DATA_BLOCK "GDB_ActiveRecipe"   // DB24
TITLE = Active recipes (Modules D+E, dual-pallet, PSC-bound)
{ S7_Optimized_Access := 'TRUE' }
// SCARA Phase 2 Module D + E active-recipe DB (V3.0, 2026-05-23). Two pallet slots (recipe1 = LEFT, recipe2 = RIGHT), each a UDT_Recipe. PSC binds member-for-member to recipe1.* and recipe2.* from separate HMI parameter sets. Pallet selection is operator-driven via the maintained bo_ExecutePallet1 / bo_ExecutePallet2 flags (WanErXin pattern -- no auto-advance); FB_PatternAutoGen mediates the mutex, picks the active recipe, writes its config to GDB_PalletizingCmd, validates both recipes independently, and latches per-pallet bo_PalletNFull alarms on cycle completion attributed to the IN-FLIGHT pallet (snapshotted at cycle start, so mid-cycle operator swaps cannot mis-attribute). Operator swaps pallets by clearing one flag and setting the other -- the just-emptied side's full bit auto-clears so it can be re-used. V3.0 also adds explicit per-pallet bo_AckPalletNFull reset bits and the bo_BothPalletsFull aggregate for HMI / future module integration.
// stored: MemoryReserve 100
   VAR
      recipe1 : "UDT_Recipe";   // Active recipe for PALLET 1 (LEFT). PSC binds and writes here from the HMI's pallet-1 parameter set. FB_PatternAutoGen consumes this each scan iff recipe1.bo_Valid is TRUE AND i16_ActivePalletIdx = 1. StartValues = the verified 16-box 4x(2x2) Module D default.
      recipe2 : "UDT_Recipe";   // Active recipe for PALLET 2 (RIGHT). PSC binds and writes here from the HMI's pallet-2 parameter set. FB_PatternAutoGen consumes this each scan iff recipe2.bo_Valid is TRUE AND i16_ActivePalletIdx = 2. StartValues match recipe1 (pallets share a default product); operator overrides via PSC if pallet 2 should carry a different box product.
      bo_PatternValid1 : Bool;   // FB_PatternAutoGen status for PALLET 1: recipe1 passed validation and its computed grid is mathematically valid. HMI lamp. (Independent of whether pallet 1 is currently active.)
      bo_PatternValid2 : Bool;   // FB_PatternAutoGen status for PALLET 2: recipe2 passed validation.
      bo_PatternError1 : Bool;   // FB_PatternAutoGen status for PALLET 1: recipe1 failed validation. HMI alarm.
      bo_PatternError2 : Bool;   // FB_PatternAutoGen status for PALLET 2: recipe2 failed validation.
      i16_ComputedGridColsX1 : Int;   // FB_PatternAutoGen echo for PALLET 1: auto-fitted columns along X.
      i16_ComputedGridColsX2 : Int;   // FB_PatternAutoGen echo for PALLET 2: auto-fitted columns along X.
      i16_ComputedGridRowsY1 : Int;   // FB_PatternAutoGen echo for PALLET 1: auto-fitted rows along Y.
      i16_ComputedGridRowsY2 : Int;   // FB_PatternAutoGen echo for PALLET 2: auto-fitted rows along Y.
      i16_ComputedBoxCount1 : Int;   // FB_PatternAutoGen echo for PALLET 1: total boxes = Cols x Rows x LayerCount. Must stay within the GDB_PalletizingPath.aCmd[] ceiling (22) or recipe1 is rejected.
      i16_ComputedBoxCount2 : Int;   // FB_PatternAutoGen echo for PALLET 2: total boxes. Same ceiling.
      bo_ExecutePallet1 : Bool := TRUE;   // Operator flag (HMI MAINTAINED button) -- "execute pallet 1" (WanErXin pattern). Setting TRUE while bo_ExecutePallet2=FALSE selects pallet 1 as active; FB_PatternAutoGen then writes recipe1 into GDB_PalletizingCmd. Cleared TRUE by operator releasing the button OR auto-cleared by FB when bo_Pallet1Full (operator must press the other side's button to swap, which auto-clears the just-emptied pallet's full bit so it can be re-used).
      bo_ExecutePallet2 : Bool := FALSE;   // Operator flag -- "execute pallet 2". Mirror of bo_ExecutePallet1 for the right-side pallet. Both flags simultaneously TRUE = mutex stalemate (FB keeps the current active pallet); both FALSE = i16_ActivePalletIdx := 0, no pallet active, GDB_PalletizingCmd left at safe defaults.
      i16_ActivePalletIdx : Int;   // FB_PatternAutoGen status: which pallet is currently active. 1 = pallet 1 (LEFT), 2 = pallet 2 (RIGHT), 0 = neither (no operator flag set OR active recipe invalid). HMI display.
      bo_Pallet1Full : Bool;   // Latched "pallet 1 full" alarm. Set TRUE by FB_PatternAutoGen when GDB_PalletizingCmd.bo_PalletDone is TRUE while i16_ActivePalletIdx = 1 (the cycle just placed the last box of pallet 1). Cleared automatically when the operator switches to pallet 2 (bo_ExecutePallet1 := FALSE AND bo_ExecutePallet2 := TRUE) -- which is interpreted as "I have emptied pallet 1, ready to re-use it later". HMI lamp/alarm.
      bo_Pallet2Full : Bool;   // Latched "pallet 2 full" alarm. Same logic as bo_Pallet1Full, mirrored.
      bo_AckPallet1Full : Bool;   // V3.0 (2026-05-23): Operator acknowledge / explicit reset for bo_Pallet1Full. HMI MAINTAINED button. While TRUE, FB_PatternAutoGen forces bo_Pallet1Full := FALSE every scan -- explicit reset path used when operator has physically emptied pallet 1 and wants to re-use it WITHOUT first having to swap to pallet 2. (The WanErXin swap-clear path remains as a convenience: pressing pallet 2's button while pallet 1's full bit is latched still clears it.) Operator releases the Ack button before re-starting the cycle so the next bo_PalletDone can re-latch bo_Pallet1Full normally.
      bo_AckPallet2Full : Bool;   // V3.0: Operator acknowledge / explicit reset for bo_Pallet2Full. Mirror of bo_AckPallet1Full.
      bo_BothPalletsFull : Bool;   // V3.0: FB-computed aggregate = bo_Pallet1Full AND bo_Pallet2Full. Single status bit for HMI / future Module F-G integration to gate "both pallets need unloading, robot should idle". Read-only from HMI side -- FB_PatternAutoGen is sole writer.
   END_VAR
BEGIN
   recipe1.sName := 'Pallet 1 Default 4x2x2';
   recipe1.bo_Valid := TRUE;
   recipe1.product.lr_Length := 400.0;
   recipe1.product.lr_Width := 600.0;
   recipe1.product.lr_Height := 200.0;
   recipe1.product.lr_Gap := 0.0;
   recipe1.pallet.lr_BaseLength := 800.0;
   recipe1.pallet.lr_BaseWidth := 1200.0;
   recipe1.pallet.i16_LayerCount := 4;
   recipe1.dynamics.lr_Velocity := 2000.0;
   recipe1.dynamics.lr_Acceleration := 10000.0;
   recipe1.dynamics.lr_Deceleration := 10000.0;
   recipe1.dynamics.lr_Jerk := 100000.0;
   recipe2.sName := 'Pallet 2 Default 4x2x2';
   recipe2.bo_Valid := TRUE;
   recipe2.product.lr_Length := 400.0;
   recipe2.product.lr_Width := 600.0;
   recipe2.product.lr_Height := 200.0;
   recipe2.product.lr_Gap := 0.0;
   recipe2.pallet.lr_BaseLength := 800.0;
   recipe2.pallet.lr_BaseWidth := 1200.0;
   recipe2.pallet.i16_LayerCount := 4;
   recipe2.dynamics.lr_Velocity := 2000.0;
   recipe2.dynamics.lr_Acceleration := 10000.0;
   recipe2.dynamics.lr_Deceleration := 10000.0;
   recipe2.dynamics.lr_Jerk := 100000.0;
END_DATA_BLOCK

DATA_BLOCK "GDB_MovePath"   // DB21
{ S7_Optimized_Access := 'TRUE' }
// stored: MemoryReserve 100
BEGIN
END_DATA_BLOCK

DATA_BLOCK "GDB_TeachCmd"   // DB27
TITLE = Teach mode commands + status (Module F)
{ S7_Optimized_Access := 'TRUE' }
// SCARA Phase 2 Module F teach-mode command + status DB (2026-05-23). HMI writes the mode toggle, per-slot operations (Capture/Verify/Clear/ClearAll), and replay controls (Start/Stop/Vel). FB_TeachCtrl reads them, executes via the shared GDB_AxisCtrl interface, and publishes back i16_TeachStep / i16_ReplayIdx / bo_ReplayDone for HMI display. Mode mutex: bo_Mode must be TRUE while GDB_MachineCmd.bo_Mode (transitional), GDB_PalletizingCmd.bo_Mode, and GDB_ManualCmd.bo_Mode are all FALSE.
// stored: MemoryReserve 100
   VAR
      bo_Mode : Bool := FALSE;   // HMI: Teach mode selector (the 4th mutex mode). TRUE = teach commands + jog active and the replay FSM can run. FALSE = ignored. Mutex with GDB_MachineCmd.bo_Mode (ABCDE, transitional -- to be deleted), GDB_PalletizingCmd.bo_Mode (palletizing), GDB_ManualCmd.bo_Mode (manual). FB_TeachCtrl REGION Mode_Gate enforces single-mode-active via statTeachOK.
      bo_ESTOP_LOCK : Bool := TRUE;   // Safety: E-Stop chain healthy (TRUE = OK, FALSE = E-Stop active). Mirrors GDB_PalletizingCmd / GDB_ManualCmd convention. Default TRUE (PLCSIM phantom; real fieldbus E-Stop integration is a separate task).
      i16_SlotIdx : Int := 1;   // HMI: which teach slot (1..16) the operator is currently operating on. Used by all four edge-pulsed operations (Capture, Verify, Clear) and as the HMI's "table row selector". Validated by FB_TeachCtrl as 1 <= idx <= 16; out-of-range pulses are ignored. Default 1.
      bo_Capture : Bool;   // HMI PULSE: capture current TCP into aPoints[i16_SlotIdx]. Edge-detected by FB_TeachCtrl. On rising edge (and only while statTeachOK = TRUE AND idx in range): reads GDB_AxisCtrl.LKinCtrl.output.actualposition (populated by FB_AxisCtrl MirrorTCP from ScaraArm3D.Position[..]), writes to aPoints[idx].position[0..3] (4..5 zeroed), sets abCaptured[idx] := TRUE, sets i16_TeachStep := 10 briefly for HMI feedback. Operator's main teach action.
      bo_Verify : Bool;   // HMI PULSE: move robot to aPoints[i16_SlotIdx]. Edge-detected. On rising edge: copies aPoints[idx].position to GDB_AxisCtrl.LKinCtrl.input.movelinear.targetposition, sets r64_velocity to lr_ReplayVel, pulses bo_execute. Used to validate that a captured slot points where the operator intended.
      bo_Clear : Bool;   // HMI PULSE: clear aPoints[i16_SlotIdx] (zero the position fields) and set abCaptured[idx] := FALSE. Edge-detected. Operator re-arms the slot for capture.
      bo_ClearAll : Bool;   // HMI PULSE: clear ALL 16 slots in one pass. Edge-detected. FB loops 1..16 clearing both aPoints[i] and abCaptured[i]. Operator's "wipe and start over" gesture.
      bo_StartReplay : Bool;   // HMI PULSE: start once-through replay of all captured slots in index order. Edge-detected. FB_TeachCtrl Replay_FSM transitions from idle (0) to load_next_slot (100), iterates aPoints[1..16] skipping uncaptured slots, drives each via the shared movelinear interface. Replay ends with bo_ReplayDone := TRUE and FSM back to idle.
      bo_StopReplay : Bool;   // HMI PULSE: abort replay immediately. Edge-detected. FB_TeachCtrl Replay_FSM transitions to idle (0) from any active state, clears bo_execute, the current move aborts via the MC layer's bo_commandaborted.
      lr_ReplayVel : LReal := 200.0;   // HMI: replay-move velocity (mm/s). Applied uniformly to every replay move and to bo_Verify moves. Default 200.0 mm/s (matches FB_ManualCtrl's safe-jog Cartesian dynamic). Auto-cycle palletizing uses 300+ mm/s.
      i16_TeachStep : Int;   // FB status: current step in FB_TeachCtrl Operator_Actions / Replay_FSM. Values: 0=idle, 10=capture-pulse-handled, 20=verify-in-flight, 30=clear-applied, 100=replay-running (i16_ReplayIdx advancing), 200=replay-done (latched until next StartReplay), 800=fault. HMI status display.
      i16_ReplayIdx : Int;   // FB status: which slot is currently being executed during replay (1..16). 0 when idle. HMI highlights the active row in the teach-table view.
      bo_ReplayDone : Bool;   // FB status: latched TRUE when replay reaches the end of captured slots (once-through). Cleared on next bo_StartReplay rising edge or on mode exit. HMI displays as a "Replay complete" lamp.
   END_VAR
BEGIN
END_DATA_BLOCK

DATA_BLOCK "GDB_TeachPoints"   // DB26
TITLE = Teach-point storage (Module F, 16 slots)
{ S7_Optimized_Access := 'TRUE' }
// SCARA Phase 2 Module F teach-point storage (V1.1, 2026-05-23). 16 slots, each carrying BOTH Cartesian TCP (aPoints[i] = LKinCtrl_typePoint, Siemens-canonical) AND joint angles (aJointAngles[i] = Array[1..4] of LReal for J1-J4). V1.1 added joint capture per Phase 2 spec §7.1 ("捕获脉冲 → 当前 TCP/关节 写点表"). Operator captures both in one bo_Capture pulse via FB_TeachCtrl. Replay (bo_StartReplay) currently walks aPoints via Cartesian linear moves; joint-space PTP replay using aJointAngles is reserved for a future extension.
// stored: MemoryReserve 100
   VAR
      aPoints : Array[1..16] of "LKinCtrl_typePoint";   // Module F teach-point slots (1..16) -- CARTESIAN. Each slot reuses the Siemens-canonical LKinCtrl_typePoint UDT: name (WString), position[0..5] LReal (Cartesian X/Y/Z/A/B/C in WCS; SCARA populates [0..3] only), coordSystem USInt (default 0=WCS), linkConstellation DWord, turnJoint[0..5] DInt. FB_TeachCtrl writes here on operator's bo_Capture edge from GDB_AxisCtrl.LKinCtrl.output.actualposition. Replay (bo_StartReplay) walks these via Cartesian linear moves.
      aJointAngles : Array[1..16, 1..4] of LReal;   // V1.1 (2026-05-23, joint extension per Phase 2 §7.1 spec "TCP/关节"): Per-slot joint angles J1/J2/J3/J4 captured at the same scan as aPoints[i]. 2D array (S7-1500T does not allow nested Array-of-Array in interface declarations -- same convention LKinCtrl_FrameTransTool's rotation matrices use). Access: aJointAngles[slot, joint] e.g. aJointAngles[3, 1] = slot 3's J1. FB_TeachCtrl writes from "ScaraArm3D".AxesData.A[1..4].Position on the same bo_Capture rising edge. Stored for archival + future joint-space PTP replay (currently replay is Cartesian-linear only). J1/J2/J4 in degrees, J3 in mm (prismatic Z per the SCARA TO config).
      abCaptured : Array[1..16] of Bool;   // Per-slot "this slot has been captured" flag. FB_TeachCtrl sets TRUE on bo_Capture rising edge for slot i16_SlotIdx (one set covers BOTH aPoints[idx] and aJointAngles[idx], V1.1); clears on bo_Clear or bo_ClearAll. Replay (bo_StartReplay) skips slots where this is FALSE. Default FALSE (no slots captured at boot).
      i16_PointCount : Int;   // FB-computed status: COUNT of TRUE bits in abCaptured[1..16]. HMI displays as "Captured slots: N / 16". Also used by FB_TeachCtrl Replay_FSM as the bound for the slot iteration (replay only runs slots where abCaptured = TRUE).
   END_VAR
BEGIN
END_DATA_BLOCK

ORGANIZATION_BLOCK "Main"   // OB1, LAD, ProgramCycle
TITLE = "Main Program Sweep (Cycle)"
{ S7_Optimized_Access := 'TRUE' }
// stored: SetENOAutomatically false
   VAR_INPUT
      Initial_Call : Bool;   // Initial call of this OB
      Remanence : Bool;   // =True, if remanent data are available
   END_VAR
BEGIN
END_ORGANIZATION_BLOCK

ORGANIZATION_BLOCK "CyclicInterrupt_10ms"   // OB30, LAD, CyclicInterrupt
{ S7_Optimized_Access := 'TRUE' }
// stored: SetENOAutomatically false
   VAR_INPUT
      Initial_Call : Bool;   // Initial call of this OB
      Event_Count : Int;   // Events discarded
   END_VAR
BEGIN
END_ORGANIZATION_BLOCK

ORGANIZATION_BLOCK "Startup"
TITLE = "Complete Restart"
{ S7_Optimized_Access := 'TRUE' }
VERSION : 1.0
// =====================================================================
// SCARA ABCDE â€” Startup (OB100)
//
// 2026-05-17 â€” Minimal startup for ABCDE 5-point demo.
// Initializes GDB_Control arrays so retain-memory drift can never zero
// them (defense pattern proven in v9, see Memory MEMORY.md â†’ cfg-retain
// fix). Clears command bits so warm-start can't replay an in-flight cmd.
//
// All HMI cmd bits live in GDB_MachineCmd (initialized via Member
// StartValue attributes in the XML â€” bo_Mode and bo_ESTOP_LOCK both
// default TRUE so an operator can immediately start). i16_AutoStep
// defaults to 0 (idle) which is the safe state.
// =====================================================================
   VAR_TEMP 
      i : Int;
   END_VAR


BEGIN
	
	 REGION Set_GroupPower_StartStopMode_defaults
	     // LKinCtrl_MC_GroupPower reads GDB_Control.StartMode[i] / StopMode[i].
	     // If any element is 0 on cold start / warm-start retain drift, MC_Power
	     // silently refuses to assert axesEnabled  - busy stuck FALSE forever.
	     // Set all 6 elements of both arrays to 1 (position-controlled enable /
	     // standard immediate-stop) on every PLC startup.
	     FOR #i := 1 TO 6 DO
	         "GDB_AxisCtrl".LKinCtrl.input.configuration.power.startMode[#i] := 1;   // 1 = enable position-controlled
	         "GDB_AxisCtrl".LKinCtrl.input.configuration.power.stopMode[#i]  := 1;   // 1 = immediate stop
	     END_FOR;
	 END_REGION
	
	 REGION Set_GroupHome_defaults
	     // LKinCtrl_MC_GroupHome reads GDB_Control.HomePos[i] / HomeMode[i].
	     // HomeMode=7 ("set actual position") is used in the SCARA demo so
	     // no physical homing motion is needed  - the operator clicks Home
	     // and the current TO joint position becomes the home reference.
	     //
	     // HomePos values per kinematic-axis index (A1=J1 base, A2=J3 z,
	     // A3=J2 elbow, A4=J4 wrist) match the SCARA3D zero pose. Indexes
	     // 5/6 (B/C orientation) unused in this 4-DOF kinematic.
	     "GDB_AxisCtrl".LKinCtrl.input.configuration.home.r64_homeposition[1] := 0.0;   // A1 = J1 base shoulder
	     "GDB_AxisCtrl".LKinCtrl.input.configuration.home.r64_homeposition[2] := 0.0;   // A2 = J3 prismatic z
	     "GDB_AxisCtrl".LKinCtrl.input.configuration.home.r64_homeposition[3] := 0.0;   // A3 = J2 elbow
	     "GDB_AxisCtrl".LKinCtrl.input.configuration.home.r64_homeposition[4] := 0.0;   // A4 = J4 wrist
	     "GDB_AxisCtrl".LKinCtrl.input.configuration.home.r64_homeposition[5] := 0.0;   // unused
	     "GDB_AxisCtrl".LKinCtrl.input.configuration.home.r64_homeposition[6] := 0.0;   // unused
	     FOR #i := 1 TO 6 DO
	         "GDB_AxisCtrl".LKinCtrl.input.configuration.home.i16_mode[#i] := 7;   // 7 = set actual position (no motion)
	     END_FOR;
	 END_REGION
	
	 REGION Set_GroupReset_RestartMode_defaults
	     // LKinCtrl_MC_GroupReset reads GDB_Control.RestartMode[1..7] of Bool.
	     // All FALSE = standard reset (clear axis error, do not re-initialize TO).
	     FOR #i := 1 TO 7 DO
	         "GDB_AxisCtrl".LKinCtrl.input.configuration.reset.restart[#i] := FALSE;
	     END_FOR;
	 END_REGION
	
	 REGION Clear_group_motion_command_bits
	     // Defensive: clear group enable/home/reset bits so warm-start can't
	     // replay an in-flight command. Operator must re-click Enable on HMI.
	     "GDB_AxisCtrl".LKinCtrl.input.bo_enable := FALSE;
	     "GDB_AxisCtrl".LKinCtrl.input.bo_reset  := FALSE;
	     "GDB_AxisCtrl".LKinCtrl.input.bo_home   := FALSE;
	 END_REGION
	
	 REGION Clear_AutoCtrl_command_bits
	     // Wang Shuo pattern: i16_AutoStep is the master state. 0 = idle.
	     // On warm-start, retain may have left step=80 (mid-cycle). Force
	     // back to 0 so operator must explicitly re-Start.
	     "GDB_MachineCmd".i16_AutoStep := 0;
	     "GDB_MachineCmd".bo_PathInitialed := FALSE;  // operator must re-init
	     "GDB_MachineCmd".bo_Alarm := FALSE;
	 END_REGION
	
	 REGION Clear_PalletizingCtrl_command_bits
	     // C69 Phase 2.2 (2026-05-18): defensively clear all palletizing-mode
	     // command bits + i16_PalletStep so warm-start can't replay a partial
	     // cycle. bo_Mode + bo_ESTOP_LOCK keep their XML StartValues (FALSE + TRUE).
	     // bo_PalletInitialed cleared - operator must re-pulse bo_InitPallet on
	     // session start to repopulate pts[] (path table is in iDB statics, not
	     // retain, so it would be all-zeros after memory reset anyway).
	     "GDB_PalletizingCmd".bo_InitPallet := FALSE;
	     "GDB_PalletizingCmd".bo_Start := FALSE;
	     "GDB_PalletizingCmd".bo_Stop := FALSE;
	     "GDB_PalletizingCmd".bo_PalletInitialed := FALSE;
	     "GDB_PalletizingCmd".bo_Alarm := FALSE;
	     "GDB_PalletizingCmd".i16_PalletStep := 0;
	 END_REGION
	
	 REGION Clear_ManualCtrl_command_bits
	     // Phase G (C67, 2026-05-18): defensively clear all manual-mode
	     // command bits so warm-start can't replay a held jog button or
	     // a latched Enable/Home/Reset. Operator must re-press on HMI.
	     // bo_Mode + bo_ESTOP_LOCK keep their XML StartValues (FALSE + TRUE).
	     "GDB_ManualCmd".bo_J1_Enable := FALSE;
	     "GDB_ManualCmd".bo_J2_Enable := FALSE;
	     "GDB_ManualCmd".bo_J3_Enable := FALSE;
	     "GDB_ManualCmd".bo_J4_Enable := FALSE;
	     "GDB_ManualCmd".bo_J1_Home := FALSE;
	     "GDB_ManualCmd".bo_J2_Home := FALSE;
	     "GDB_ManualCmd".bo_J3_Home := FALSE;
	     "GDB_ManualCmd".bo_J4_Home := FALSE;
	     "GDB_ManualCmd".bo_J1_Reset := FALSE;
	     "GDB_ManualCmd".bo_J2_Reset := FALSE;
	     "GDB_ManualCmd".bo_J3_Reset := FALSE;
	     "GDB_ManualCmd".bo_J4_Reset := FALSE;
	     "GDB_ManualCmd".bo_J1_JogForward := FALSE;
	     "GDB_ManualCmd".bo_J1_JogBackward := FALSE;
	     "GDB_ManualCmd".bo_J2_JogForward := FALSE;
	     "GDB_ManualCmd".bo_J2_JogBackward := FALSE;
	     "GDB_ManualCmd".bo_J3_JogForward := FALSE;
	     "GDB_ManualCmd".bo_J3_JogBackward := FALSE;
	     "GDB_ManualCmd".bo_J4_JogForward := FALSE;
	     "GDB_ManualCmd".bo_J4_JogBackward := FALSE;
	     "GDB_ManualCmd".bo_KinEnable := FALSE;
	     "GDB_ManualCmd".bo_KinHome := FALSE;
	     "GDB_ManualCmd".bo_KinReset := FALSE;
	     "GDB_ManualCmd".bo_KinGo := FALSE;
	     // cfgKinTarget{X,Y,Z,A} keep their XML StartValues (A-point safe defaults).
	 END_REGION
	
	
END_ORGANIZATION_BLOCK

FUNCTION_BLOCK "FB_HMIStatusMirror"
{ S7_Optimized_Access := 'TRUE' }
VERSION : 0.1
// =====================================================================
// SCARA ABCDE Phase 2.4 (C71, 2026-05-18) â€” HMI Read-Only Facade Mirror
//
// Consolidates ~35 display tags from across the system into GDB_HMI_Status
// each OB1 scan. HMI binds to GDB_HMI_Status for ALL READS (single binding
// surface); HMI continues to write directly to the per-mode cmd DBs
// (GDB_MachineCmd / GDB_PalletizingCmd / GDB_ManualCmd) for commands.
//
// 5 REGIONs:
//   REGION 1: Active-mode arbitration (compute 0=None/1=ABCDE/2=Pallet/3=Manual)
//   REGION 2: Mode-routed currentStep + totalSteps + target XYZA
//   REGION 3: Group axis status (axesEnabled/Homed/Error/Ready)
//   REGION 4: Per-joint status (4 joints Ã— 6 fields = 24 assignments)
//   REGION 5: Safety + cycle-init flags + diagnostics
//
// Per-scan cost: ~35 simple assignments + 1 IF/ELSIF chain. Negligible
// vs the FB_AutoCtrl_ABCDE / FB_AutoCtrl_Palletizing 4-REGION machinery.
//
// Placement in Main.scl: LAST in the FB call sequence so all upstream
// FBs (FB_AxisCtrl, FB_ManualCtrl, FB_AutoCtrl_ABCDE, FB_AutoCtrl_Palletizing,
// FB_MCDDataTransfer) have written their fresh state by the time this
// FB reads + mirrors them.
//
// Mutex semantics: arbitration uses IF/ELSIF priority chain (ABCDE wins
// over Palletizing wins over Manual when multiple modes are TRUE).
// PLC's REAL mutex enforcement is at each FB's START gate (silent reject
// of conflicting Start pulses). This activeMode field is a DISPLAY-LAYER
// derivative â€” operator should rely on it to know "which cycle is
// actually running", but write-coordination is HMI's job (per C70 Â§4).
// =====================================================================
   VAR_TEMP 
      tempActiveMode : Int;
   END_VAR


BEGIN
	
	
	 // =====================================================================
	 // REGION 1 â€” Active-mode arbitration
	 // Priority: ABCDE > Palletizing > Manual > None
	 // Only one bo_Mode should be TRUE at a time (HMI's responsibility per
	 // C70 Â§4 Option 4A); but if multiple are set, priority chain picks one
	 // for display. PLC's per-FB START gates enforce the real mutex.
	 // =====================================================================
	 IF "GDB_MachineCmd".bo_Mode THEN
	     #tempActiveMode := 1;       // ABCDE
	 ELSIF "GDB_PalletizingCmd".bo_Mode THEN
	     #tempActiveMode := 2;       // Palletizing
	 ELSIF "GDB_ManualCmd".bo_Mode THEN
	     #tempActiveMode := 3;       // Manual
	 ELSE
	     #tempActiveMode := 0;       // None / Idle
	 END_IF;
	 "GDB_HMI_Status".activeMode := #tempActiveMode;
	
	 // =====================================================================
	 // REGION 2 â€” Mode-routed currentStep + totalSteps + target XYZA
	 // ABCDE mode: step from i16_AutoStep, total=5, target from ABCDE iDB
	 // Palletizing mode: step from i16_PalletStep, total=48, target from Pal iDB
	 // Manual mode: step=0, total=0, target HOLDS last value (no write)
	 // None: step=0, total=0, target holds last value
	 // =====================================================================
	 CASE #tempActiveMode OF
	     1: // ABCDE
	         "GDB_HMI_Status".currentStep := "GDB_MachineCmd".i16_AutoStep;
	         "GDB_HMI_Status".totalSteps := 5;
	         "GDB_HMI_Status".target_x := "instFB_AutoCtrl_ABCDE".statTargetPos.x;
	         "GDB_HMI_Status".target_y := "instFB_AutoCtrl_ABCDE".statTargetPos.y;
	         "GDB_HMI_Status".target_z := "instFB_AutoCtrl_ABCDE".statTargetPos.z;
	         "GDB_HMI_Status".target_a := "instFB_AutoCtrl_ABCDE".statTargetPos.a;
	     2: // Palletizing
	         "GDB_HMI_Status".currentStep := "GDB_PalletizingCmd".i16_PalletStep;
	         "GDB_HMI_Status".totalSteps := 48;
	         "GDB_HMI_Status".target_x := "instFB_AutoCtrl_Palletizing".statTargetPos.x;
	         "GDB_HMI_Status".target_y := "instFB_AutoCtrl_Palletizing".statTargetPos.y;
	         "GDB_HMI_Status".target_z := "instFB_AutoCtrl_Palletizing".statTargetPos.z;
	         "GDB_HMI_Status".target_a := "instFB_AutoCtrl_Palletizing".statTargetPos.a;
	     3: // Manual â€” no auto-target trajectory; show 0 steps
	         "GDB_HMI_Status".currentStep := 0;
	         "GDB_HMI_Status".totalSteps := 0;
	         // target_x/y/z/a NOT written â€” preserves last commanded target value
	     ELSE // None / Idle
	         "GDB_HMI_Status".currentStep := 0;
	         "GDB_HMI_Status".totalSteps := 0;
	         // target stays at last value
	 END_CASE;
	
	 // =====================================================================
	 // REGION 3 â€” Group axis status
	 // =====================================================================
	 "GDB_HMI_Status".axesEnabled := "GDB_Control".axesEnabled;
	 "GDB_HMI_Status".axesHomed := "GDB_Control".axesHomed;
	 "GDB_HMI_Status".axesError := "GDB_Control".axesError;
	 "GDB_HMI_Status".axesReady := "GDB_Control".axesReady;
	
	 // =====================================================================
	 // REGION 4 â€” Per-joint status (4 joints Ã— 6 fields = 24 assignments)
	 // Reads bool fields from GDB_ManualStatus (FB_ManualCtrl REGION 5 mirror),
	 // and reads actual position/velocity direct from J{n}_SCARA_Arm3D TO.
	 // Joint-name convention throughout (no kinematic-group swap on HMI surface).
	 // =====================================================================
	 "GDB_HMI_Status".j1_enabled := "GDB_ManualStatus".bo_J1_Enabled;
	 "GDB_HMI_Status".j1_homed := "GDB_ManualStatus".bo_J1_Homed;
	 "GDB_HMI_Status".j1_error := "GDB_ManualStatus".bo_J1_Error;
	 "GDB_HMI_Status".j1_jogActive := "GDB_ManualStatus".bo_J1_JogActive;
	 "GDB_HMI_Status".j1_actualPos := "J1_SCARA_Arm3D".ActualPosition;
	 "GDB_HMI_Status".j1_actualVel := "J1_SCARA_Arm3D".ActualVelocity;
	
	 "GDB_HMI_Status".j2_enabled := "GDB_ManualStatus".bo_J2_Enabled;
	 "GDB_HMI_Status".j2_homed := "GDB_ManualStatus".bo_J2_Homed;
	 "GDB_HMI_Status".j2_error := "GDB_ManualStatus".bo_J2_Error;
	 "GDB_HMI_Status".j2_jogActive := "GDB_ManualStatus".bo_J2_JogActive;
	 "GDB_HMI_Status".j2_actualPos := "J2_SCARA_Arm3D".ActualPosition;
	 "GDB_HMI_Status".j2_actualVel := "J2_SCARA_Arm3D".ActualVelocity;
	
	 "GDB_HMI_Status".j3_enabled := "GDB_ManualStatus".bo_J3_Enabled;
	 "GDB_HMI_Status".j3_homed := "GDB_ManualStatus".bo_J3_Homed;
	 "GDB_HMI_Status".j3_error := "GDB_ManualStatus".bo_J3_Error;
	 "GDB_HMI_Status".j3_jogActive := "GDB_ManualStatus".bo_J3_JogActive;
	 "GDB_HMI_Status".j3_actualPos := "J3_SCARA_Arm3D".ActualPosition;
	 "GDB_HMI_Status".j3_actualVel := "J3_SCARA_Arm3D".ActualVelocity;
	
	 "GDB_HMI_Status".j4_enabled := "GDB_ManualStatus".bo_J4_Enabled;
	 "GDB_HMI_Status".j4_homed := "GDB_ManualStatus".bo_J4_Homed;
	 "GDB_HMI_Status".j4_error := "GDB_ManualStatus".bo_J4_Error;
	 "GDB_HMI_Status".j4_jogActive := "GDB_ManualStatus".bo_J4_JogActive;
	 "GDB_HMI_Status".j4_actualPos := "J4_SCARA_Arm3D".ActualPosition;
	 "GDB_HMI_Status".j4_actualVel := "J4_SCARA_Arm3D".ActualVelocity;
	
	 // =====================================================================
	 // REGION 5 â€” Safety + cycle-init flags + diagnostics
	 // =====================================================================
	 "GDB_HMI_Status".estopLock := "GDB_MachineCmd".bo_ESTOP_LOCK;
	 "GDB_HMI_Status".alarm := "GDB_MachineCmd".bo_Alarm OR "GDB_PalletizingCmd".bo_Alarm;
	 "GDB_HMI_Status".pathInitialed := "GDB_MachineCmd".bo_PathInitialed;
	 "GDB_HMI_Status".palletInitialed := "GDB_PalletizingCmd".bo_PalletInitialed;
	 "GDB_HMI_Status".toolActive := "instFB_AxisCtrl".statToolActivated;
	
	
END_FUNCTION_BLOCK

FUNCTION_BLOCK "FB_MCDDataTransfer"
{ S7_Optimized_Access := 'TRUE' }
VERSION : 0.2
// =====================================================================
// FB_MCDDataTransfer rev 0.2 (2026-05-17 Phase C.0)
//
// CHANGES vs rev 0.1:
//   - ADDED 8 explicit-named direct-from-TO_Axis assignments after the
//     existing kinematic-group FOR loop:
//       GDB_MCDData.J{1..4}_{ActualPosition, ActualVelocity} :=
//         J{1..4}_SCARA_Arm3D.{ActualPosition, ActualVelocity};
//
// RATIONALE: TO_Axis tags (J{n}_SCARA_Arm3D.ActualPosition + ActualVelocity)
// are NOT exposed via PLCSIM-Adv API directly (returns Error -4 DoesNotExist).
// HMI runtime reads them fine via TIA's S7 driver (HMI agent's TIA Compile
// passed 0E/0W against those bindings per CompileGreen handoff). For
// PLCSIM-Adv API monitoring + future tooling parity, mirror them to
// explicit-named GDB members.
//
// The existing kinematic-group FOR loop (Position[1..4] + Velocity[1..4])
// stays for back-compat with NX MCD signal adapter consumers + existing
// smoke-test code.
//
// HMI binding strategy is UNCHANGED — HMI continues to read TO_Axis direct
// via S7 driver (per HMI agent's UBP design). The new GDB members are
// PLC-side diagnostic mirror only, NOT a new HMI surface.
// =====================================================================
   VAR_TEMP 
      tempIndex : Int;
   END_VAR


BEGIN
	// Kinematic-group view of per-axis data (rev 0.1, preserved for back-compat):
	FOR #tempIndex := 1 TO 4 DO
	
	    "GDB_MCDData".Position[#tempIndex] := "ScaraArm3D".AxesData.A[#tempIndex].Position;
	
	    "GDB_MCDData".Velocity[#tempIndex] := "ScaraArm3D".AxesData.A[#tempIndex].Velocity;
	END_FOR;
	
	// === Phase C.0 (rev 0.2) — explicit-named direct-from-TO_Axis mirror ===
	// Closes PLCSIM-Adv API gap for TO_Axis tag access. HMI runtime still
	// reads TO_Axis direct via S7 driver; these mirror fields exist for
	// PLCSIM-Adv API / future tooling parity. See FB header comment.
	"GDB_MCDData".J1_ActualPosition := "J1_SCARA_Arm3D".ActualPosition;
	"GDB_MCDData".J1_ActualVelocity := "J1_SCARA_Arm3D".ActualVelocity;
	"GDB_MCDData".J2_ActualPosition := "J2_SCARA_Arm3D".ActualPosition;
	"GDB_MCDData".J2_ActualVelocity := "J2_SCARA_Arm3D".ActualVelocity;
	"GDB_MCDData".J3_ActualPosition := "J3_SCARA_Arm3D".ActualPosition;
	"GDB_MCDData".J3_ActualVelocity := "J3_SCARA_Arm3D".ActualVelocity;
	"GDB_MCDData".J4_ActualPosition := "J4_SCARA_Arm3D".ActualPosition;
	"GDB_MCDData".J4_ActualVelocity := "J4_SCARA_Arm3D".ActualVelocity;
	
END_FUNCTION_BLOCK

FUNCTION_BLOCK "FB_AutoCtrl_5Pts"
{ S7_Optimized_Access := 'TRUE' }
VERSION : 1.2
// =====================================================================
// SCARA ABCDE - 5-Point Auto Cycle  (Phase 4a, 2026-05-21)
//
// Huashili-pattern CASE state machine. Runs in OB1 (process logic). It
// owns the ABCDE 5-point sequence and commands motion ONLY by writing
// GDB_AxisCtrl.LKinCtrl.input.movelinear - it never calls an MC
// instruction. FB_AxisCtrl (OB30) runs the actual MC_MoveLinearAbsolute.
//
// Structure (Huashili FB_AutoCtrl): the REGIONs Initialise path / startup
// / Pause / Stop / Alarm / E_Stop edge-detect the HMI command bits and
// jump the step variable; REGION Auto holds the CASE.
//
// Step model (GDB_MachineCmd.i16_AutoStep):
//   0   idle              10  head reset       20  preconditions
//   30  load target       50  issue motion     75  pause hold
//   100 wait-in-place     110 handshake done   200 abort
//   230 advance / wrap    800 E-Stop hold      900 tail reset
//
// Move handshake (cross-OB, OB1<->OB30): step 50 holds bo_execute TRUE;
// step 100 waits output.movelinear.bo_done; step 110 then waits bo_done
// to clear - this confirms FB_AxisCtrl saw bo_execute drop, so the next
// move is a clean rising edge for MC_MoveLinearAbsolute.
//
// Replaces FB_AutoCtrl_ABCDE (retired once this FB is verified).
//
// V1.2 (2026-05-22) - R6: REGION Pause + CASE step 75 implement the auto-cycle
// pause. bo_Pause (edge) halts the cycle mid-move via FB_AxisCtrl's
// MC_GroupInterrupt; resume on the Start edge. Stop / E-Stop override.
// V1.1 (2026-05-22) - step 30 sets input.movelinear.bo_isPTP := FALSE so the
// ABCDE square always uses Cartesian linear moves. FB_AxisCtrl V2.3 added a
// PTP route on that shared bit (for the palletizing transits); ABCDE opts out.
// =====================================================================
   VAR
      pts : Array[1..5] of "UDT_typePoint5";
      statTargetPos { S7_SetPoint := 'False' } : "UDT_typePoint5";
      statPointIdx : Int;
      sRTRIGInitPath {InstructionName := 'R_TRIG'; LibVersion := '1.0'} : R_TRIG;
      sRTRIGStart {InstructionName := 'R_TRIG'; LibVersion := '1.0'} : R_TRIG;
      sRTRIGStop {InstructionName := 'R_TRIG'; LibVersion := '1.0'} : R_TRIG;
      sRTRIGAlarm {InstructionName := 'R_TRIG'; LibVersion := '1.0'} : R_TRIG;
      sRTRIGPause {InstructionName := 'R_TRIG'; LibVersion := '1.0'} : R_TRIG;
      statStepBeforePause : Int;   // step to resume to after a pause (R6)
   END_VAR


BEGIN

    REGION Initialise path
        // On the HMI Init-Path rising edge, build the ABCDE 5-point table -
        // a square in the WCS, all at Z = 400 mm. (Ported from FB_AutoCtrl_ABCDE.)
        #sRTRIGInitPath(CLK := "GDB_MachineCmd".bo_InitPath);
        IF #sRTRIGInitPath.Q THEN
            #pts[1].x := 1800.0; #pts[1].y := 0.0;    #pts[1].z := 400.0; #pts[1].a := 0.0;   // A
            #pts[2].x := 1800.0; #pts[2].y := 300.0;  #pts[2].z := 400.0; #pts[2].a := 0.0;   // B
            #pts[3].x := 1500.0; #pts[3].y := 300.0;  #pts[3].z := 400.0; #pts[3].a := 0.0;   // C
            #pts[4].x := 1500.0; #pts[4].y := -300.0; #pts[4].z := 400.0; #pts[4].a := 0.0;   // D
            #pts[5].x := 1800.0; #pts[5].y := -300.0; #pts[5].z := 400.0; #pts[5].a := 0.0;   // E
            "GDB_MachineCmd".bo_PathInitialed := TRUE;
        END_IF;
    END_REGION


    REGION startup
        // Start permissive: AUTO mode, E-Stop healthy, idle, path initialised,
        // no alarm. On the Start rising edge, enter the cycle at head reset.
        #sRTRIGStart(CLK := "GDB_MachineCmd".bo_Start);
        IF "GDB_MachineCmd".bo_Mode
            AND "GDB_MachineCmd".bo_ESTOP_LOCK
            AND ("GDB_MachineCmd".i16_AutoStep = 0)
            AND #sRTRIGStart.Q
            AND "GDB_MachineCmd".bo_PathInitialed
            AND NOT "GDB_MachineCmd".bo_Alarm
        THEN
            "GDB_MachineCmd".i16_AutoStep := 10;
        END_IF;
    END_REGION


    REGION Pause
        // R6 - auto-cycle pause. On the bo_Pause rising edge, while the cycle
        // is running, save the current step, raise the halt request to the
        // 600 axis layer (FB_AxisCtrl runs MC_GroupInterrupt - the SCARA halts
        // mid-trajectory, axes stay enabled), and jump to the pause-hold step
        // 75. Resume is handled in step 75. Stop / E-Stop (later REGIONs)
        // override Pause - they re-target step 200 / 800 from step 75.
        #sRTRIGPause(CLK := "GDB_MachineCmd".bo_Pause);
        IF "GDB_MachineCmd".bo_Mode
            AND "GDB_MachineCmd".bo_ESTOP_LOCK
            AND #sRTRIGPause.Q
            AND NOT "GDB_MachineCmd".bo_Alarm
            AND ("GDB_MachineCmd".i16_AutoStep >= 10)
            AND ("GDB_MachineCmd".i16_AutoStep <= 230)
            AND ("GDB_MachineCmd".i16_AutoStep <> 75)
        THEN
            #statStepBeforePause := "GDB_MachineCmd".i16_AutoStep;
            "GDB_AxisCtrl".LKinCtrl.input.bo_movepathhalt := TRUE;
            "GDB_MachineCmd".i16_AutoStep := 75;
        END_IF;
    END_REGION


    REGION Stop
        // Stop -> abort. Route through step 200 so the in-flight move command
        // is dropped and the tail reset (900) runs before returning to idle.
        #sRTRIGStop(CLK := "GDB_MachineCmd".bo_Stop);
        IF #sRTRIGStop.Q
            AND ("GDB_MachineCmd".i16_AutoStep >= 10)
            AND ("GDB_MachineCmd".i16_AutoStep <= 230)
        THEN
            "GDB_MachineCmd".i16_AutoStep := 200;
        END_IF;
    END_REGION


    REGION Alarm
        // Any system alarm -> abort (same path as Stop).
        #sRTRIGAlarm(CLK := "GDB_MachineCmd".bo_Alarm);
        IF #sRTRIGAlarm.Q
            AND ("GDB_MachineCmd".i16_AutoStep >= 10)
            AND ("GDB_MachineCmd".i16_AutoStep <= 230)
        THEN
            "GDB_MachineCmd".i16_AutoStep := 200;
        END_IF;
    END_REGION


    REGION E_Stop
        // E-Stop chain open (bo_ESTOP_LOCK = FALSE) -> jump to the hold
        // state 800 from any running step.
        IF NOT "GDB_MachineCmd".bo_ESTOP_LOCK
            AND ("GDB_MachineCmd".i16_AutoStep >= 10)
            AND ("GDB_MachineCmd".i16_AutoStep <= 230)
        THEN
            "GDB_MachineCmd".i16_AutoStep := 800;
        END_IF;
    END_REGION


    REGION Auto

        CASE "GDB_MachineCmd".i16_AutoStep OF

            0:  // Idle - await Start
                ;

            10: // Head reset - clear the in-flight move command, reset index
                "GDB_AxisCtrl".LKinCtrl.input.movelinear.bo_execute := FALSE;
                #statPointIdx := 1;
                "GDB_MachineCmd".i16_AutoStep := 20;

            20: // Preconditions - wait until the OB30 axis layer is ready
                //                  (axes enabled + homed + no fault)
                IF "GDB_AxisCtrl".LKinCtrl.output.bo_ready THEN
                    "GDB_MachineCmd".i16_AutoStep := 30;
                END_IF;

            30: // Path-data assignment - load pts[idx] into the move command.
                // Parameters BEFORE command: target + dynamics set here; the
                // execute bit is set only in step 50.
                #statTargetPos := #pts[#statPointIdx];
                "GDB_AxisCtrl".LKinCtrl.input.movelinear.targetposition.x := #statTargetPos.x;
                "GDB_AxisCtrl".LKinCtrl.input.movelinear.targetposition.y := #statTargetPos.y;
                "GDB_AxisCtrl".LKinCtrl.input.movelinear.targetposition.z := #statTargetPos.z;
                "GDB_AxisCtrl".LKinCtrl.input.movelinear.targetposition.a := #statTargetPos.a;
                "GDB_AxisCtrl".LKinCtrl.input.movelinear.targetposition.b := 0.0;
                "GDB_AxisCtrl".LKinCtrl.input.movelinear.targetposition.c := 0.0;
                "GDB_AxisCtrl".LKinCtrl.input.movelinear.r64_velocity     := 300.0;
                "GDB_AxisCtrl".LKinCtrl.input.movelinear.r64_acceleration := 3000.0;
                "GDB_AxisCtrl".LKinCtrl.input.movelinear.r64_deceleration := 3000.0;
                "GDB_AxisCtrl".LKinCtrl.input.movelinear.r64_jerk         := 30000.0;
                // ABCDE square stays Cartesian linear (no base-crossing path).
                "GDB_AxisCtrl".LKinCtrl.input.movelinear.bo_isPTP         := FALSE;
                "GDB_MachineCmd".i16_AutoStep := 50;

            50: // Issue motion - hand the move to the 600 axis layer
                "GDB_AxisCtrl".LKinCtrl.input.movelinear.bo_execute := TRUE;
                "GDB_MachineCmd".i16_AutoStep := 100;

            75: // Pause hold (R6) - the cycle is frozen here. The SCARA holds
                // position (FB_AxisCtrl ran MC_GroupInterrupt; axes stay
                // enabled). bo_execute is held, so the interrupted move keeps
                // its command for a clean resume. Resume on the Start rising
                // edge: release the halt request and return to the step the
                // pause interrupted.
                IF #sRTRIGStart.Q THEN
                    "GDB_AxisCtrl".LKinCtrl.input.bo_movepathhalt := FALSE;
                    "GDB_MachineCmd".i16_AutoStep := #statStepBeforePause;
                END_IF;

            100: // Wait-in-place - FB_AxisCtrl reports the move complete.
                 // On error / abort, bail to the abort step.
                IF "GDB_AxisCtrl".LKinCtrl.output.movelinear.bo_done THEN
                    "GDB_AxisCtrl".LKinCtrl.input.movelinear.bo_execute := FALSE;
                    "GDB_MachineCmd".i16_AutoStep := 110;
                ELSIF "GDB_AxisCtrl".LKinCtrl.output.movelinear.bo_error
                    OR "GDB_AxisCtrl".LKinCtrl.output.movelinear.bo_commandaborted
                THEN
                    "GDB_AxisCtrl".LKinCtrl.input.movelinear.bo_execute := FALSE;
                    "GDB_MachineCmd".i16_AutoStep := 200;
                END_IF;

            110: // Handshake done - wait for bo_done to clear, confirming the
                 // OB30 axis layer saw bo_execute drop. Guarantees the next
                 // move is a clean rising edge for MC_MoveLinearAbsolute.
                IF NOT "GDB_AxisCtrl".LKinCtrl.output.movelinear.bo_done THEN
                    "GDB_MachineCmd".i16_AutoStep := 230;
                END_IF;

            200: // Abort - planned group stop, then tail reset. Raise
                 // bo_movepathstop so FB_AxisCtrl's MC_GroupStop halts the move
                 // mid-trajectory; drop the command + pause request; advance to
                 // the tail reset once the stop concludes (or the group faults).
                "GDB_AxisCtrl".LKinCtrl.input.movelinear.bo_execute := FALSE;
                "GDB_AxisCtrl".LKinCtrl.input.bo_movepathhalt := FALSE;
                "GDB_AxisCtrl".LKinCtrl.input.bo_movepathstop := TRUE;
                IF "GDB_AxisCtrl".LKinCtrl.output.bo_stopped
                    OR "GDB_AxisCtrl".LKinCtrl.output.bo_fault
                THEN
                    "GDB_MachineCmd".i16_AutoStep := 900;
                END_IF;

            230: // Advance - next point; the ABCDE cycle wraps E -> A
                IF #statPointIdx >= 5 THEN
                    #statPointIdx := 1;
                ELSE
                    #statPointIdx := #statPointIdx + 1;
                END_IF;
                "GDB_MachineCmd".i16_AutoStep := 30;

            800: // E-Stop hold - command + pause request dropped, planned stop
                 // raised; auto-recovers to the tail reset once the E-Stop chain
                 // is healthy again.
                "GDB_AxisCtrl".LKinCtrl.input.movelinear.bo_execute := FALSE;
                "GDB_AxisCtrl".LKinCtrl.input.bo_movepathhalt := FALSE;
                "GDB_AxisCtrl".LKinCtrl.input.bo_movepathstop := TRUE;
                IF "GDB_MachineCmd".bo_ESTOP_LOCK THEN
                    "GDB_MachineCmd".i16_AutoStep := 900;
                END_IF;

            900: // Tail reset - mirror of step 10; clears the planned-stop
                 // request and returns to idle
                "GDB_AxisCtrl".LKinCtrl.input.movelinear.bo_execute := FALSE;
                "GDB_AxisCtrl".LKinCtrl.input.bo_movepathstop := FALSE;
                #statPointIdx := 1;
                "GDB_MachineCmd".i16_AutoStep := 0;

            ELSE  // Unknown step - fail safe to idle
                "GDB_AxisCtrl".LKinCtrl.input.movelinear.bo_execute := FALSE;
                "GDB_MachineCmd".i16_AutoStep := 0;

        END_CASE;

    END_REGION

END_FUNCTION_BLOCK

FUNCTION_BLOCK "FB_AutoCtrl_ABCDE"
{ S7_Optimized_Access := 'TRUE' }
VERSION : 2.1
// =====================================================================
// SCARA ABCDE 5-Point Continuous Auto Cycle
// (2026-05-17 rev 2.1 — fixed invalid per-element Position[i] := assignment)
//
// CHANGES vs v2.0:
//   - Position parameter to MC_MoveLinearAbsolute: changed from per-element
//     `Position[1] := ..., Position[2] := ...` (which TIA V20 SCL rejects)
//     to whole-array `Position := #tempPosArray` per the proven v9 pattern
//     in FB_TestRawMoveLinAbs.scl line 45
//
// CHANGES vs v1.0 (backed up at .backup/2026-05-17/500_AutoCtrl/):
//   - Step pattern: 11-state → 6-state per source spec §3.3
//   - Removed LKinCtrl-dependent permissive per source spec line 11
//
// Wang Shuo / Huashili 4-REGION pattern (source spec §3.3+§3.5):
//   REGION 1: 初始化路径 / INITIALIZE_PATH
//   REGION 2: 启动 / START                — permissive AND → step:=10
//   REGION 3: 停止 / STOP                 — R_TRIG → step:=0
//   REGION 4: 自动 / AUTO main CASE       — 6 states (0/10/20/30/40/50)
//     0=idle, 10=去A, 20=去B, 30=去C, 40=去D, 50=去E (cycle wrap 50→10)
//
// ONE shared instMoveLinAbs (multi-instance) re-triggered per step on
// rising-edge of step change. KEY to avoiding v9's OB91 overflow.
// =====================================================================

   VAR
      // === Edge-detect instances (Wang Shuo pattern) ===
      sRTRIGInitialPath { S7_SetPoint := 'False' } : R_TRIG;
      sRTRIGStart       { S7_SetPoint := 'False' } : R_TRIG;
      sRTRIGStop        { S7_SetPoint := 'False' } : R_TRIG;

      // === Motion FB: ONE system MC_MoveLinearAbsolute, re-triggered per step ===
      instMoveLinAbs { InstructionName := 'MC_MOVELINEARABSOLUTE'; LibVersion := '9.0'; S7_SetPoint := 'False' } : MC_MOVELINEARABSOLUTE;

      // === 5-point hardcoded ABCDE path (set in REGION 1) ===
      pts { S7_SetPoint := 'False' } : Array[1..5] of "UDT_typePoint5";

      // === Static state ===
      statTargetPos    { ExternalWritable := 'False' } : "UDT_typePoint5";   // currently commanded target (HMI display)
      statOldStep      { S7_SetPoint := 'False' } : Int;                      // for step-change edge detection
      statMoveDoneOld  { S7_SetPoint := 'False' } : Bool;                     // for MoveLinAbs.Done rising-edge detection
      statExecutePulse { S7_SetPoint := 'False' } : Bool;                     // one-scan Execute pulse on step change
   END_VAR

   VAR_TEMP
      tempCurrentPtIdx : Int;                  // 1..5 mapping from i16_AutoStep
      tempStepChanged  : Bool;
      tempIsAutoStep   : Bool;                 // TRUE when step IN [10..50]
      tempPosArray     : Array[1..6] of LReal; // Position array for MC_MoveLinAbs call (4 used + 2 trailing zeros)
   END_VAR


BEGIN

	// =====================================================================
	// REGION 1 — INITIALIZE_PATH (source spec §2.1)
	// =====================================================================
	#sRTRIGInitialPath(CLK := "GDB_MachineCmd".bo_InitPath);
	IF #sRTRIGInitialPath.Q THEN
	    // ABCDE — square pattern in WCS, all at Z=400mm above home.
	    #pts[1].x := 1800.0;  #pts[1].y :=    0.0;  #pts[1].z := 400.0;  #pts[1].a := 0.0;   // A
	    #pts[2].x := 1800.0;  #pts[2].y :=  300.0;  #pts[2].z := 400.0;  #pts[2].a := 0.0;   // B
	    #pts[3].x := 1500.0;  #pts[3].y :=  300.0;  #pts[3].z := 400.0;  #pts[3].a := 0.0;   // C
	    #pts[4].x := 1500.0;  #pts[4].y := -300.0;  #pts[4].z := 400.0;  #pts[4].a := 0.0;   // D
	    #pts[5].x := 1800.0;  #pts[5].y := -300.0;  #pts[5].z := 400.0;  #pts[5].a := 0.0;   // E
	    "GDB_MachineCmd".bo_PathInitialed := TRUE;
	END_IF;

	// =====================================================================
	// REGION 2 — START (source spec §2.2)
	// =====================================================================
	#sRTRIGStart(CLK := "GDB_MachineCmd".bo_Start);
	IF "GDB_MachineCmd".bo_Mode
	   AND "GDB_MachineCmd".bo_ESTOP_LOCK
	   AND ("GDB_MachineCmd".i16_AutoStep = 0)
	   AND #sRTRIGStart.Q
	   AND "GDB_MachineCmd".bo_PathInitialed
	   AND NOT "GDB_MachineCmd".bo_Alarm
	THEN
	    "GDB_MachineCmd".i16_AutoStep := 10;
	END_IF;

	// =====================================================================
	// REGION 3 — STOP (source spec §2.3)
	// =====================================================================
	#sRTRIGStop(CLK := "GDB_MachineCmd".bo_Stop);
	IF #sRTRIGStop.Q THEN
	    "GDB_MachineCmd".i16_AutoStep := 0;
	END_IF;

	// =====================================================================
	// REGION 4 — AUTO main CASE (source spec §3.3, 6 states)
	// =====================================================================

	// Detect step-change for Execute pulse
	#tempStepChanged := ("GDB_MachineCmd".i16_AutoStep <> #statOldStep);
	#statOldStep := "GDB_MachineCmd".i16_AutoStep;

	// Classify current step as "active auto step" [10..50]
	#tempIsAutoStep := ("GDB_MachineCmd".i16_AutoStep >= 10)
	                   AND ("GDB_MachineCmd".i16_AutoStep <= 50);

	// Map step → point index (10→1, 20→2, 30→3, 40→4, 50→5)
	IF #tempIsAutoStep THEN
	    #tempCurrentPtIdx := "GDB_MachineCmd".i16_AutoStep / 10;
	    #statTargetPos := #pts[#tempCurrentPtIdx];
	END_IF;

	// Execute pulse: high for ONE scan when entering a new auto step
	#statExecutePulse := #tempStepChanged AND #tempIsAutoStep;

	// Build the 6-element Position array (4 used + 2 trailing zeros)
	#tempPosArray[1] := #statTargetPos.x;
	#tempPosArray[2] := #statTargetPos.y;
	#tempPosArray[3] := #statTargetPos.z;
	#tempPosArray[4] := #statTargetPos.a;
	#tempPosArray[5] := 0.0;
	#tempPosArray[6] := 0.0;

	// Drive MC_MoveLinearAbsolute on the kinematic group.
	// Raw system FB — no LKinCtrl wrapper (source spec line 11).
	// Whole-array Position passing per v9 FB_TestRawMoveLinAbs.scl line 45.
	#instMoveLinAbs(AxesGroup    := "ScaraArm3D",
	                Execute      := #statExecutePulse,
	                Position     := #tempPosArray,
	                Velocity     := 300.0,
	                Acceleration := 3000.0,
	                Deceleration := 3000.0,
	                Jerk         := 30000.0,
	                BufferMode   := 1);   // 1 = BM_BUFFERED (basic, source spec §3.4)
	                                      //     For V8 blending (Phase F): change to 5 = BM_BLENDING_HIGH

	// On MoveLinAbs.Done rising-edge in an auto step, advance to next step
	// (source spec §3.4 + §3.5 cycle wrap at step=50)
	IF #instMoveLinAbs.Done AND NOT #statMoveDoneOld AND #tempIsAutoStep THEN
	    IF "GDB_MachineCmd".i16_AutoStep = 50 THEN
	        "GDB_MachineCmd".i16_AutoStep := 10;        // cycle wrap E → A (§3.5)
	    ELSE
	        "GDB_MachineCmd".i16_AutoStep :=
	            "GDB_MachineCmd".i16_AutoStep + 10;     // 10→20→30→40→50
	    END_IF;
	END_IF;
	#statMoveDoneOld := #instMoveLinAbs.Done;

END_FUNCTION_BLOCK

FUNCTION_BLOCK "FB_AutoCtrl_Palletizing"
{ S7_Optimized_Access := 'TRUE' }
VERSION : 5.3
// =====================================================================
// SCARA Palletizing - Parameterized-Grid Auto Cycle  (Phase 4b, 2026-05-21)
//
// Huashili-pattern CASE state machine. Runs in OB1 (process logic). It
// owns the palletizing sequence and commands motion ONLY by writing
// GDB_AxisCtrl.LKinCtrl.input.movelinear - it never calls an MC
// instruction. FB_AxisCtrl (OB30) runs the MC_MoveLinearAbsolute.
//
// V5.3 (2026-05-22) - Module C: the path builder is parameterized. Box grid
// (i16_LayerCount / i16_GridRowsY / i16_GridColsX), pitches (lr_BoxPitchX/Y)
// and dynamics (lr_MoveVelocity / lr_MoveAccel / lr_MoveDecel / lr_MoveJerk)
// are GDB_PalletizingCmd config; the 16-box 4x(2x2) pattern is the StartValue
// default. Builder rewritten as one index-decomposed grid loop. Prereq for D.
// V5.2 (2026-05-22) - R6: REGION Pause + CASE step 75 add the auto-cycle pause.
// bo_Pause (edge) halts the cycle mid-move via FB_AxisCtrl's MC_GroupInterrupt
// (a gripped box stays gripped); resume on the Start edge. Stop / E-Stop override.
// V5.1 (2026-05-22) - the two pick<->place transits (cmd 2 ABOVE_PICK and
// cmd 6 APPROACH_PLACE) are now cmdType 4 = MOVE_PTP. A Cartesian linear
// transit swept the TCP on a straight line across the robot base and faulted
// the kinematics on the near-base singularity. MOVE_PTP routes (via
// FB_AxisCtrl) to MC_MoveDirectAbsolute - joint-space, no Cartesian-path
// constraint. The 4 vertical pick/place moves stay cmdType 1 = linear.
// V5.0 - rebuilt onto the Huashili 7-REGION + CASE shell (same pattern as
// FB_AutoCtrl_5Pts); motion split out to the 600 axis layer. The command-
// list builder (16 boxes x 9 commands -> GDB_PalletizingPath.aCmd) is
// carried over verbatim from V4.2 into REGION Initialise path. The V4.2
// progress-based executor is replaced by the CASE: one aCmd[] entry per
// pass, MOVE commands handed to the axis layer with an execute/done
// handshake. The CASE serializes moves (waits for bo_done) - the V4.2
// BufferMode-5 cross-command blending is traded for the clean structure.
//
// Step model (GDB_PalletizingCmd.i16_PalletStep):
//   0 idle  10 head reset  20 preconditions  30 fetch + dispatch
//   40 gripper dwell  50 issue move  60 wait arrival  65 arrival settle
//   75 pause hold  100 wait move done  110 handshake done  200 abort
//   230 cycle complete  800 E-Stop hold  900 tail reset
//
// aCmd[] command types: 0 = END  1 = MOVE (linear)  2 = GRIPPER
//   3 = WAIT_ARRIVAL  4 = MOVE_PTP (joint-space transit, base-singularity-safe).
// =====================================================================
   VAR
      sRTRIGInitialPath {InstructionName := 'R_TRIG'; LibVersion := '1.0'} : R_TRIG;
      sRTRIGStart {InstructionName := 'R_TRIG'; LibVersion := '1.0'} : R_TRIG;
      sRTRIGStop {InstructionName := 'R_TRIG'; LibVersion := '1.0'} : R_TRIG;
      sRTRIGAlarm {InstructionName := 'R_TRIG'; LibVersion := '1.0'} : R_TRIG;
      statTargetPos { S7_SetPoint := 'False' } : "UDT_typePoint5";
      statCmdPtr : Int;   // index into GDB_PalletizingPath.aCmd (0 = idle)
      statBoxesPlaced : Int;
      instGripperTimer {InstructionName := 'TON_TIME'; LibVersion := '1.0'} : TON_TIME;
      instArrivalSettleTimer {InstructionName := 'TON_TIME'; LibVersion := '1.0'} : TON_TIME;
      sRTRIGPause {InstructionName := 'R_TRIG'; LibVersion := '1.0'} : R_TRIG;
      statStepBeforePause : Int;   // step to resume to after a pause (R6)
   END_VAR

   VAR_TEMP
      tempBoxIdx : Int;     // builder - running box index 1..i16_TotalBoxes
      tempPerLayer : Int;   // builder - boxes per layer = GridRowsY * GridColsX
      tempLayer : Int;      // builder - layer 1..i16_LayerCount
      tempRow : Int;        // builder - grid row 0..i16_GridRowsY-1
      tempCol : Int;        // builder - grid col 0..i16_GridColsX-1
      tempCmdW : Int;       // builder - write cursor into aCmd
      tempPlaceZ : LReal;
      tempBoxX : LReal;
      tempBoxY : LReal;
      tempPickX : LReal;
      tempPickY : LReal;
      tempCmdType : Int;    // command type at statCmdPtr (executor)
   END_VAR


BEGIN

    REGION Initialise path
        // ================================================================
        // Command-list builder - parameterized (Module C, Phase 2 section 4).
        // Box grid + move velocity come from GDB_PalletizingCmd config:
        // i16_LayerCount / i16_GridRowsY / i16_GridColsX / lr_BoxPitchX /
        // lr_BoxPitchY / lr_MoveVelocity. 9 commands/box: WAIT_ARRIVAL,
        // ABOVE_PICK, PICK_DESCEND, GRIPPER(grip), PICK_RAISE, APPROACH_PLACE,
        // PLACE_DESCEND, GRIPPER(release), PLACE_RETRACT + one END_OF_PATH.
        // cmdType: 0=END 1=MOVE 2=GRIPPER 3=WAIT_ARRIVAL 4=MOVE_PTP.
        // Build order: bottom layer first; within a layer row-major (Y x X),
        // the grid centred on the pallet top.
        // ================================================================
        #sRTRIGInitialPath(CLK := "GDB_PalletizingCmd".bo_InitPallet);
        IF #sRTRIGInitialPath.Q THEN
            #tempPerLayer := "GDB_PalletizingCmd".i16_GridRowsY
                           * "GDB_PalletizingCmd".i16_GridColsX;
            "GDB_PalletizingCmd".i16_TotalBoxes := "GDB_PalletizingCmd".i16_LayerCount
                                                 * #tempPerLayer;
            #tempCmdW  := 0;
            #tempPickX := "GDB_PalletizingCmd".lr_PickX + "GDB_PalletizingCmd".lr_WristOffsetX;
            #tempPickY := "GDB_PalletizingCmd".lr_PickY + "GDB_PalletizingCmd".lr_WristOffsetY;

            FOR #tempBoxIdx := 1 TO "GDB_PalletizingCmd".i16_TotalBoxes DO
                // decompose the linear box index into layer / grid row / col
                #tempLayer := (#tempBoxIdx - 1) / #tempPerLayer + 1;
                #tempRow   := ((#tempBoxIdx - 1) / "GDB_PalletizingCmd".i16_GridColsX)
                              MOD "GDB_PalletizingCmd".i16_GridRowsY;
                #tempCol   := (#tempBoxIdx - 1) MOD "GDB_PalletizingCmd".i16_GridColsX;
                #tempPlaceZ := "GDB_PalletizingCmd".lr_PalletTopZ
                             + #tempLayer * "GDB_PalletizingCmd".lr_BoxHeight;
                // grid box position, centred on the pallet top
                #tempBoxX := "GDB_PalletizingCmd".lr_PalletTopX
                           + (#tempCol - ("GDB_PalletizingCmd".i16_GridColsX - 1) / 2.0)
                             * "GDB_PalletizingCmd".lr_BoxPitchX;
                #tempBoxY := "GDB_PalletizingCmd".lr_PalletTopY
                           + (#tempRow - ("GDB_PalletizingCmd".i16_GridRowsY - 1) / 2.0)
                             * "GDB_PalletizingCmd".lr_BoxPitchY;

                // cmd 1 -- WAIT_ARRIVAL
                #tempCmdW := #tempCmdW + 1;
                "GDB_PalletizingPath".aCmd[#tempCmdW].i16_CmdType := 3;
                "GDB_PalletizingPath".aCmd[#tempCmdW].i16_HmiStep := (#tempBoxIdx - 1) * 3 + 1;

                // cmd 2 -- MOVE_PTP ABOVE_PICK (transit; joint-space, base-safe)
                #tempCmdW := #tempCmdW + 1;
                "GDB_PalletizingPath".aCmd[#tempCmdW].i16_CmdType    := 4;
                "GDB_PalletizingPath".aCmd[#tempCmdW].x              := #tempPickX;
                "GDB_PalletizingPath".aCmd[#tempCmdW].y              := #tempPickY;
                "GDB_PalletizingPath".aCmd[#tempCmdW].z              := "GDB_PalletizingCmd".lr_PickZ
                                                                      + "GDB_PalletizingCmd".lr_PickApproachZOffset
                                                                      + "GDB_PalletizingCmd".lr_WristOffsetZ;
                "GDB_PalletizingPath".aCmd[#tempCmdW].a              := 0.0;
                "GDB_PalletizingPath".aCmd[#tempCmdW].lr_Velocity    := "GDB_PalletizingCmd".lr_MoveVelocity;
                "GDB_PalletizingPath".aCmd[#tempCmdW].i16_BufferMode := 5;
                "GDB_PalletizingPath".aCmd[#tempCmdW].bo_IsBoxEnd    := FALSE;
                "GDB_PalletizingPath".aCmd[#tempCmdW].i16_HmiStep    := (#tempBoxIdx - 1) * 3 + 1;

                // cmd 3 -- MOVE PICK_DESCEND (stop)
                #tempCmdW := #tempCmdW + 1;
                "GDB_PalletizingPath".aCmd[#tempCmdW].i16_CmdType    := 1;
                "GDB_PalletizingPath".aCmd[#tempCmdW].x              := #tempPickX;
                "GDB_PalletizingPath".aCmd[#tempCmdW].y              := #tempPickY;
                "GDB_PalletizingPath".aCmd[#tempCmdW].z              := "GDB_PalletizingCmd".lr_PickZ
                                                                      + "GDB_PalletizingCmd".lr_WristOffsetZ;
                "GDB_PalletizingPath".aCmd[#tempCmdW].a              := 0.0;
                "GDB_PalletizingPath".aCmd[#tempCmdW].lr_Velocity    := "GDB_PalletizingCmd".lr_MoveVelocity;
                "GDB_PalletizingPath".aCmd[#tempCmdW].i16_BufferMode := 1;
                "GDB_PalletizingPath".aCmd[#tempCmdW].bo_IsBoxEnd    := FALSE;
                "GDB_PalletizingPath".aCmd[#tempCmdW].i16_HmiStep    := (#tempBoxIdx - 1) * 3 + 1;

                // cmd 4 -- GRIPPER grip (vacuum ON, hold lr_GripperCloseMs)
                #tempCmdW := #tempCmdW + 1;
                "GDB_PalletizingPath".aCmd[#tempCmdW].i16_CmdType      := 2;
                "GDB_PalletizingPath".aCmd[#tempCmdW].lr_DwellMs       := "GDB_PalletizingCmd".lr_GripperCloseMs;
                "GDB_PalletizingPath".aCmd[#tempCmdW].bo_GripperGrip   := TRUE;
                "GDB_PalletizingPath".aCmd[#tempCmdW].bo_GripperRelease := FALSE;
                "GDB_PalletizingPath".aCmd[#tempCmdW].i16_HmiStep      := (#tempBoxIdx - 1) * 3 + 1;

                // cmd 5 -- MOVE PICK_RAISE (blend)
                #tempCmdW := #tempCmdW + 1;
                "GDB_PalletizingPath".aCmd[#tempCmdW].i16_CmdType    := 1;
                "GDB_PalletizingPath".aCmd[#tempCmdW].x              := #tempPickX;
                "GDB_PalletizingPath".aCmd[#tempCmdW].y              := #tempPickY;
                "GDB_PalletizingPath".aCmd[#tempCmdW].z              := "GDB_PalletizingCmd".lr_PickZ
                                                                      + "GDB_PalletizingCmd".lr_PickApproachZOffset
                                                                      + "GDB_PalletizingCmd".lr_WristOffsetZ;
                "GDB_PalletizingPath".aCmd[#tempCmdW].a              := 0.0;
                "GDB_PalletizingPath".aCmd[#tempCmdW].lr_Velocity    := "GDB_PalletizingCmd".lr_MoveVelocity;
                "GDB_PalletizingPath".aCmd[#tempCmdW].i16_BufferMode := 5;
                "GDB_PalletizingPath".aCmd[#tempCmdW].bo_IsBoxEnd    := FALSE;
                "GDB_PalletizingPath".aCmd[#tempCmdW].i16_HmiStep    := (#tempBoxIdx - 1) * 3 + 1;

                // cmd 6 -- MOVE_PTP APPROACH_PLACE (transit; joint-space, base-safe)
                #tempCmdW := #tempCmdW + 1;
                "GDB_PalletizingPath".aCmd[#tempCmdW].i16_CmdType    := 4;
                "GDB_PalletizingPath".aCmd[#tempCmdW].x              := #tempBoxX + "GDB_PalletizingCmd".lr_WristOffsetX;
                "GDB_PalletizingPath".aCmd[#tempCmdW].y              := #tempBoxY + "GDB_PalletizingCmd".lr_WristOffsetY;
                "GDB_PalletizingPath".aCmd[#tempCmdW].z              := #tempPlaceZ
                                                                      + "GDB_PalletizingCmd".lr_PlaceApproachZOffset
                                                                      + "GDB_PalletizingCmd".lr_WristOffsetZ;
                "GDB_PalletizingPath".aCmd[#tempCmdW].a              := 0.0;
                "GDB_PalletizingPath".aCmd[#tempCmdW].lr_Velocity    := "GDB_PalletizingCmd".lr_MoveVelocity;
                "GDB_PalletizingPath".aCmd[#tempCmdW].i16_BufferMode := 5;
                "GDB_PalletizingPath".aCmd[#tempCmdW].bo_IsBoxEnd    := FALSE;
                "GDB_PalletizingPath".aCmd[#tempCmdW].i16_HmiStep    := (#tempBoxIdx - 1) * 3 + 1;

                // cmd 7 -- MOVE PLACE_DESCEND (stop)
                #tempCmdW := #tempCmdW + 1;
                "GDB_PalletizingPath".aCmd[#tempCmdW].i16_CmdType    := 1;
                "GDB_PalletizingPath".aCmd[#tempCmdW].x              := #tempBoxX + "GDB_PalletizingCmd".lr_WristOffsetX;
                "GDB_PalletizingPath".aCmd[#tempCmdW].y              := #tempBoxY + "GDB_PalletizingCmd".lr_WristOffsetY;
                "GDB_PalletizingPath".aCmd[#tempCmdW].z              := #tempPlaceZ + "GDB_PalletizingCmd".lr_WristOffsetZ;
                "GDB_PalletizingPath".aCmd[#tempCmdW].a              := 0.0;
                "GDB_PalletizingPath".aCmd[#tempCmdW].lr_Velocity    := "GDB_PalletizingCmd".lr_MoveVelocity;
                "GDB_PalletizingPath".aCmd[#tempCmdW].i16_BufferMode := 1;
                "GDB_PalletizingPath".aCmd[#tempCmdW].bo_IsBoxEnd    := FALSE;
                "GDB_PalletizingPath".aCmd[#tempCmdW].i16_HmiStep    := (#tempBoxIdx - 1) * 3 + 2;

                // cmd 8 -- GRIPPER release (vacuum OFF + blow-off, hold lr_GripperOpenMs)
                #tempCmdW := #tempCmdW + 1;
                "GDB_PalletizingPath".aCmd[#tempCmdW].i16_CmdType      := 2;
                "GDB_PalletizingPath".aCmd[#tempCmdW].lr_DwellMs       := "GDB_PalletizingCmd".lr_GripperOpenMs;
                "GDB_PalletizingPath".aCmd[#tempCmdW].bo_GripperGrip   := FALSE;
                "GDB_PalletizingPath".aCmd[#tempCmdW].bo_GripperRelease := TRUE;
                "GDB_PalletizingPath".aCmd[#tempCmdW].i16_HmiStep      := (#tempBoxIdx - 1) * 3 + 2;

                // cmd 9 -- MOVE PLACE_RETRACT (blend) -- box end
                #tempCmdW := #tempCmdW + 1;
                "GDB_PalletizingPath".aCmd[#tempCmdW].i16_CmdType    := 1;
                "GDB_PalletizingPath".aCmd[#tempCmdW].x              := #tempBoxX + "GDB_PalletizingCmd".lr_WristOffsetX;
                "GDB_PalletizingPath".aCmd[#tempCmdW].y              := #tempBoxY + "GDB_PalletizingCmd".lr_WristOffsetY;
                "GDB_PalletizingPath".aCmd[#tempCmdW].z              := #tempPlaceZ
                                                                      + "GDB_PalletizingCmd".lr_PlaceApproachZOffset
                                                                      + "GDB_PalletizingCmd".lr_WristOffsetZ;
                "GDB_PalletizingPath".aCmd[#tempCmdW].a              := 0.0;
                "GDB_PalletizingPath".aCmd[#tempCmdW].lr_Velocity    := "GDB_PalletizingCmd".lr_MoveVelocity;
                "GDB_PalletizingPath".aCmd[#tempCmdW].i16_BufferMode := 5;
                "GDB_PalletizingPath".aCmd[#tempCmdW].bo_IsBoxEnd    := TRUE;
                "GDB_PalletizingPath".aCmd[#tempCmdW].i16_HmiStep    := (#tempBoxIdx - 1) * 3 + 3;
            END_FOR;

            // END_OF_PATH terminator
            #tempCmdW := #tempCmdW + 1;
            "GDB_PalletizingPath".aCmd[#tempCmdW].i16_CmdType := 0;
            "GDB_PalletizingPath".i16_CmdCount := #tempCmdW;

            "GDB_PalletizingCmd".bo_PalletInitialed := TRUE;
            "GDB_PalletizingCmd".bo_PalletDone := FALSE;
        END_IF;
    END_REGION


    REGION startup
        // Start permissive: palletizing AUTO mode, E-Stop healthy, idle,
        // path initialised, no alarm, AND the 3-way mode mutex (ABCDE +
        // manual both off). On the Start rising edge, enter at head reset.
        #sRTRIGStart(CLK := "GDB_PalletizingCmd".bo_Start);
        IF "GDB_PalletizingCmd".bo_Mode
            AND "GDB_PalletizingCmd".bo_ESTOP_LOCK
            AND ("GDB_PalletizingCmd".i16_PalletStep = 0)
            AND #sRTRIGStart.Q
            AND "GDB_PalletizingCmd".bo_PalletInitialed
            AND NOT "GDB_PalletizingCmd".bo_Alarm
            AND NOT "GDB_MachineCmd".bo_Mode
            AND NOT "GDB_ManualCmd".bo_Mode
        THEN
            "GDB_PalletizingCmd".i16_PalletStep := 10;
        END_IF;
    END_REGION


    REGION Pause
        // R6 - auto-cycle pause. On the bo_Pause rising edge, while the cycle
        // is running, save the current step, raise the halt request to the
        // 600 axis layer (FB_AxisCtrl runs MC_GroupInterrupt - the SCARA halts
        // mid-trajectory, axes stay enabled, a gripped box stays gripped), and
        // jump to the pause-hold step 75. Resume is handled in step 75. Stop /
        // E-Stop (later REGIONs) override Pause from step 75.
        #sRTRIGPause(CLK := "GDB_PalletizingCmd".bo_Pause);
        IF "GDB_PalletizingCmd".bo_Mode
            AND "GDB_PalletizingCmd".bo_ESTOP_LOCK
            AND #sRTRIGPause.Q
            AND NOT "GDB_PalletizingCmd".bo_Alarm
            AND ("GDB_PalletizingCmd".i16_PalletStep >= 10)
            AND ("GDB_PalletizingCmd".i16_PalletStep <= 230)
            AND ("GDB_PalletizingCmd".i16_PalletStep <> 75)
        THEN
            #statStepBeforePause := "GDB_PalletizingCmd".i16_PalletStep;
            "GDB_AxisCtrl".LKinCtrl.input.bo_movepathhalt := TRUE;
            "GDB_PalletizingCmd".i16_PalletStep := 75;
        END_IF;
    END_REGION


    REGION Stop
        // Stop -> abort. Route through step 200 so the in-flight move command
        // and the gripper outputs are dropped and the tail reset (900) runs.
        #sRTRIGStop(CLK := "GDB_PalletizingCmd".bo_Stop);
        IF #sRTRIGStop.Q
            AND ("GDB_PalletizingCmd".i16_PalletStep >= 10)
            AND ("GDB_PalletizingCmd".i16_PalletStep <= 230)
        THEN
            "GDB_PalletizingCmd".i16_PalletStep := 200;
        END_IF;
    END_REGION


    REGION Alarm
        // Any palletizing alarm -> abort (same path as Stop).
        #sRTRIGAlarm(CLK := "GDB_PalletizingCmd".bo_Alarm);
        IF #sRTRIGAlarm.Q
            AND ("GDB_PalletizingCmd".i16_PalletStep >= 10)
            AND ("GDB_PalletizingCmd".i16_PalletStep <= 230)
        THEN
            "GDB_PalletizingCmd".i16_PalletStep := 200;
        END_IF;
    END_REGION


    REGION E_Stop
        // E-Stop chain open (bo_ESTOP_LOCK = FALSE) -> jump to the hold
        // state 800 from any running step.
        IF NOT "GDB_PalletizingCmd".bo_ESTOP_LOCK
            AND ("GDB_PalletizingCmd".i16_PalletStep >= 10)
            AND ("GDB_PalletizingCmd".i16_PalletStep <= 230)
        THEN
            "GDB_PalletizingCmd".i16_PalletStep := 800;
        END_IF;
    END_REGION


    REGION Auto

        CASE "GDB_PalletizingCmd".i16_PalletStep OF

            0:  // Idle - await Start
                ;

            10: // Head reset - clear command + gripper outputs, reset pointers
                "GDB_AxisCtrl".LKinCtrl.input.movelinear.bo_execute := FALSE;
                "GDB_MCDData".bo_gripperGrip    := FALSE;
                "GDB_MCDData".bo_gripperRelease := FALSE;
                #statCmdPtr      := 1;
                #statBoxesPlaced := 0;
                "GDB_PalletizingCmd".bo_PalletDone := FALSE;
                "GDB_PalletizingCmd".i16_PalletStep := 20;

            20: // Preconditions - wait until the OB30 axis layer is ready
                IF "GDB_AxisCtrl".LKinCtrl.output.bo_ready THEN
                    "GDB_PalletizingCmd".i16_PalletStep := 30;
                END_IF;

            30: // Fetch + dispatch the command at statCmdPtr.
                // The aCmd[] read is nested inside the bounds IF - S7-1500 SCL
                // does not guarantee short-circuit evaluation.
                IF #statCmdPtr >= 1 AND #statCmdPtr <= 200 THEN
                    #tempCmdType := "GDB_PalletizingPath".aCmd[#statCmdPtr].i16_CmdType;
                    CASE #tempCmdType OF
                        0:  // END_OF_PATH -> cycle complete
                            "GDB_PalletizingCmd".i16_PalletStep := 230;

                        1, 4:  // MOVE (1 = linear, 4 = PTP transit) - load target + dynamics
                            #statTargetPos.x := "GDB_PalletizingPath".aCmd[#statCmdPtr].x;
                            #statTargetPos.y := "GDB_PalletizingPath".aCmd[#statCmdPtr].y;
                            #statTargetPos.z := "GDB_PalletizingPath".aCmd[#statCmdPtr].z;
                            #statTargetPos.a := "GDB_PalletizingPath".aCmd[#statCmdPtr].a;
                            "GDB_AxisCtrl".LKinCtrl.input.movelinear.targetposition.x := #statTargetPos.x;
                            "GDB_AxisCtrl".LKinCtrl.input.movelinear.targetposition.y := #statTargetPos.y;
                            "GDB_AxisCtrl".LKinCtrl.input.movelinear.targetposition.z := #statTargetPos.z;
                            "GDB_AxisCtrl".LKinCtrl.input.movelinear.targetposition.a := #statTargetPos.a;
                            "GDB_AxisCtrl".LKinCtrl.input.movelinear.targetposition.b := 0.0;
                            "GDB_AxisCtrl".LKinCtrl.input.movelinear.targetposition.c := 0.0;
                            "GDB_AxisCtrl".LKinCtrl.input.movelinear.r64_velocity     := "GDB_PalletizingPath".aCmd[#statCmdPtr].lr_Velocity;
                            "GDB_AxisCtrl".LKinCtrl.input.movelinear.r64_acceleration := "GDB_PalletizingCmd".lr_MoveAccel;
                            "GDB_AxisCtrl".LKinCtrl.input.movelinear.r64_deceleration := "GDB_PalletizingCmd".lr_MoveDecel;
                            "GDB_AxisCtrl".LKinCtrl.input.movelinear.r64_jerk         := "GDB_PalletizingCmd".lr_MoveJerk;
                            // route the move: linear (cmdType 1) or PTP transit (cmdType 4)
                            "GDB_AxisCtrl".LKinCtrl.input.movelinear.bo_isPTP := (#tempCmdType = 4);
                            "GDB_PalletizingCmd".i16_PalletStep := 50;

                        2:  // GRIPPER - write the suction-cup level bits
                            "GDB_MCDData".bo_gripperGrip    := "GDB_PalletizingPath".aCmd[#statCmdPtr].bo_GripperGrip;
                            "GDB_MCDData".bo_gripperRelease := "GDB_PalletizingPath".aCmd[#statCmdPtr].bo_GripperRelease;
                            "GDB_PalletizingCmd".i16_PalletStep := 40;

                        3:  // WAIT_ARRIVAL
                            "GDB_PalletizingCmd".i16_PalletStep := 60;

                        ELSE  // unknown command type -> abort
                            "GDB_PalletizingCmd".i16_PalletStep := 200;
                    END_CASE;
                ELSE
                    "GDB_PalletizingCmd".i16_PalletStep := 200;   // pointer out of range
                END_IF;

            40: // Gripper dwell - hold the grip/release for lr_DwellMs
                IF #statCmdPtr >= 1 AND #statCmdPtr <= 200 THEN
                    #instGripperTimer(IN := TRUE,
                                      PT := DINT_TO_TIME(LREAL_TO_DINT("GDB_PalletizingPath".aCmd[#statCmdPtr].lr_DwellMs)));
                    IF #instGripperTimer.Q THEN
                        #instGripperTimer(IN := FALSE, PT := T#0MS);
                        "GDB_MCDData".bo_gripperRelease := FALSE;   // end any blow-off pulse
                        #statCmdPtr := #statCmdPtr + 1;
                        "GDB_PalletizingCmd".i16_PalletStep := 30;
                    END_IF;
                ELSE
                    "GDB_PalletizingCmd".i16_PalletStep := 200;
                END_IF;

            50: // Issue motion - hand the move to the 600 axis layer
                "GDB_AxisCtrl".LKinCtrl.input.movelinear.bo_execute := TRUE;
                "GDB_PalletizingCmd".i16_PalletStep := 100;

            60: // Wait arrival - gate the pick on box arrival. Real mode waits
                // for the PalletizingSensor LEVEL; phantom mode (no sensor
                // gate) proceeds at once.
                IF "GDB_MCDData".PalletizingSensor
                    OR NOT "GDB_PalletizingCmd".bo_RequireSensorGate
                THEN
                    "GDB_PalletizingCmd".i16_PalletStep := 65;
                END_IF;

            65: // Arrival settle - let the box settle before descend-to-pick
                #instArrivalSettleTimer(IN := TRUE,
                                        PT := DINT_TO_TIME(LREAL_TO_DINT("GDB_PalletizingCmd".lr_ArrivalSettleMs)));
                IF #instArrivalSettleTimer.Q THEN
                    #instArrivalSettleTimer(IN := FALSE, PT := T#0MS);
                    #statCmdPtr := #statCmdPtr + 1;
                    "GDB_PalletizingCmd".i16_PalletStep := 30;
                END_IF;

            75: // Pause hold (R6) - the cycle is frozen here. The SCARA holds
                // position (FB_AxisCtrl ran MC_GroupInterrupt; axes stay
                // enabled) and a gripped box stays gripped. bo_execute is held
                // so an interrupted move keeps its command for a clean resume.
                // Resume on the Start rising edge: release the halt request and
                // return to the step the pause interrupted.
                IF #sRTRIGStart.Q THEN
                    "GDB_AxisCtrl".LKinCtrl.input.bo_movepathhalt := FALSE;
                    "GDB_PalletizingCmd".i16_PalletStep := #statStepBeforePause;
                END_IF;

            100: // Wait-in-place - FB_AxisCtrl reports the move complete.
                 // On error / abort, bail to the abort step.
                IF "GDB_AxisCtrl".LKinCtrl.output.movelinear.bo_done THEN
                    "GDB_AxisCtrl".LKinCtrl.input.movelinear.bo_execute := FALSE;
                    "GDB_PalletizingCmd".i16_PalletStep := 110;
                ELSIF "GDB_AxisCtrl".LKinCtrl.output.movelinear.bo_error
                    OR "GDB_AxisCtrl".LKinCtrl.output.movelinear.bo_commandaborted
                THEN
                    "GDB_AxisCtrl".LKinCtrl.input.movelinear.bo_execute := FALSE;
                    "GDB_PalletizingCmd".i16_PalletStep := 200;
                END_IF;

            110: // Handshake done - wait for bo_done to clear (the OB30 axis
                 // layer saw bo_execute drop), count a box on a box-end move,
                 // then advance the command pointer.
                IF NOT "GDB_AxisCtrl".LKinCtrl.output.movelinear.bo_done THEN
                    IF #statCmdPtr >= 1 AND #statCmdPtr <= 200 THEN
                        IF "GDB_PalletizingPath".aCmd[#statCmdPtr].bo_IsBoxEnd THEN
                            #statBoxesPlaced := #statBoxesPlaced + 1;
                        END_IF;
                    END_IF;
                    #statCmdPtr := #statCmdPtr + 1;
                    "GDB_PalletizingCmd".i16_PalletStep := 30;
                END_IF;

            200: // Abort - planned group stop, then tail reset. Raise
                 // bo_movepathstop so FB_AxisCtrl's MC_GroupStop halts the move
                 // mid-trajectory; drop the command, pause request and gripper
                 // outputs; advance to the tail reset once the stop concludes
                 // (or the group is already faulted).
                "GDB_AxisCtrl".LKinCtrl.input.movelinear.bo_execute := FALSE;
                "GDB_AxisCtrl".LKinCtrl.input.bo_movepathhalt := FALSE;
                "GDB_AxisCtrl".LKinCtrl.input.bo_movepathstop := TRUE;
                "GDB_MCDData".bo_gripperGrip    := FALSE;
                "GDB_MCDData".bo_gripperRelease := FALSE;
                IF "GDB_AxisCtrl".LKinCtrl.output.bo_stopped
                    OR "GDB_AxisCtrl".LKinCtrl.output.bo_fault
                THEN
                    "GDB_PalletizingCmd".i16_PalletStep := 900;
                END_IF;

            230: // Cycle complete - all boxes placed (END_OF_PATH reached)
                "GDB_PalletizingCmd".bo_PalletDone := TRUE;
                "GDB_AxisCtrl".LKinCtrl.input.movelinear.bo_execute := FALSE;
                "GDB_MCDData".bo_gripperGrip    := FALSE;
                "GDB_MCDData".bo_gripperRelease := FALSE;
                "GDB_PalletizingCmd".i16_PalletStep := 0;

            800: // E-Stop hold - outputs + pause request dropped, planned stop
                 // raised; auto-recovers to the tail reset once the E-Stop chain
                 // is healthy again.
                "GDB_AxisCtrl".LKinCtrl.input.movelinear.bo_execute := FALSE;
                "GDB_AxisCtrl".LKinCtrl.input.bo_movepathhalt := FALSE;
                "GDB_AxisCtrl".LKinCtrl.input.bo_movepathstop := TRUE;
                "GDB_MCDData".bo_gripperGrip    := FALSE;
                "GDB_MCDData".bo_gripperRelease := FALSE;
                IF "GDB_PalletizingCmd".bo_ESTOP_LOCK THEN
                    "GDB_PalletizingCmd".i16_PalletStep := 900;
                END_IF;

            900: // Tail reset - mirror of step 10; clears the planned-stop
                 // request and returns to idle
                "GDB_AxisCtrl".LKinCtrl.input.movelinear.bo_execute := FALSE;
                "GDB_AxisCtrl".LKinCtrl.input.bo_movepathstop := FALSE;
                "GDB_MCDData".bo_gripperGrip    := FALSE;
                "GDB_MCDData".bo_gripperRelease := FALSE;
                #statCmdPtr := 0;
                "GDB_PalletizingCmd".i16_PalletStep := 0;

            ELSE  // Unknown step - fail safe to idle
                "GDB_AxisCtrl".LKinCtrl.input.movelinear.bo_execute := FALSE;
                "GDB_MCDData".bo_gripperGrip    := FALSE;
                "GDB_MCDData".bo_gripperRelease := FALSE;
                "GDB_PalletizingCmd".i16_PalletStep := 0;

        END_CASE;

    END_REGION

END_FUNCTION_BLOCK

FUNCTION_BLOCK "FB_AxisCtrl"
{ S7_Optimized_Access := 'TRUE' }
VERSION : 1.1
// =====================================================================
// Per-axis enable / home / reset for SCARA 4-joint kinematic
// (2026-05-17 rev 1.1 — fixed invalid MC_GROUPRESET reference)
//
// CHANGES vs v1.0:
//   - REPLACED `MC_GROUPRESET` (NOT a valid TIA V20 system instruction —
//     verified by reading LKinCtrl_MC_GroupReset.scl in .backup/2026-05-17/:
//     it uses MC_RESET per-axis + MC_RESET on the TO_Kinematics)
//   - Now uses 4× per-axis MC_RESET + 1× MC_RESET on ScaraArm3D kinematic TO
//
// PURPOSE: Replaces LKinCtrl_MC_GroupPower / GroupHome / GroupReset wrappers
// (in .backup/2026-05-17/) with raw system MC instructions per source spec
// line 11 ("不用任何的库" / no libraries).
//
// PER-SCAN MC INSTRUCTION COUNT:
//   - 4× MC_Power (one per joint J1..J4)
//   - 4× MC_Home  (one per joint J1..J4)
//   - 5× MC_Reset (4 per joint + 1 on kinematic TO — LKinCtrl pattern)
//   Total: 13 declared, ~4-5 actively pulsing at any time. Plus
//   FB_AutoCtrl_ABCDE's 1× MC_MoveLinearAbsolute = ~5-6 active MC slots
//   vs v9's ~50 actively pulsing → OB91 headroom preserved.
//
// HMI bindings (via GDB_Control):
//   enableAxes (W Bool)   → MC_Power.Enable for all 4 joints
//   resetAxes  (W Bool)   → MC_Reset.Execute for all 4 joints + kin TO
//   homeAxes   (W Bool)   → MC_Home.Execute for all 4 joints (single rising-edge)
//
// Mirror outputs to GDB_Control:
//   axesEnabled := AND of all 4 MC_Power.Status
//   axesHomed   := AND of all 4 MC_Home.Done
//   axesError   := OR of all errors (Power + Home + Reset)
// =====================================================================

   VAR
      // === Multi-instance MC_Power per joint axis ===
      instPower_J1 { InstructionName := 'MC_POWER'; LibVersion := '9.0' } : MC_POWER;
      instPower_J2 { InstructionName := 'MC_POWER'; LibVersion := '9.0' } : MC_POWER;
      instPower_J3 { InstructionName := 'MC_POWER'; LibVersion := '9.0' } : MC_POWER;
      instPower_J4 { InstructionName := 'MC_POWER'; LibVersion := '9.0' } : MC_POWER;

      // === Multi-instance MC_Home per joint axis ===
      instHome_J1 { InstructionName := 'MC_HOME'; LibVersion := '9.0' } : MC_HOME;
      instHome_J2 { InstructionName := 'MC_HOME'; LibVersion := '9.0' } : MC_HOME;
      instHome_J3 { InstructionName := 'MC_HOME'; LibVersion := '9.0' } : MC_HOME;
      instHome_J4 { InstructionName := 'MC_HOME'; LibVersion := '9.0' } : MC_HOME;

      // === Multi-instance MC_Reset per joint axis + kinematic TO ===
      // (per LKinCtrl_MC_GroupReset pattern at .backup line 38-39)
      instReset_J1  { InstructionName := 'MC_RESET'; LibVersion := '9.0' } : MC_RESET;
      instReset_J2  { InstructionName := 'MC_RESET'; LibVersion := '9.0' } : MC_RESET;
      instReset_J3  { InstructionName := 'MC_RESET'; LibVersion := '9.0' } : MC_RESET;
      instReset_J4  { InstructionName := 'MC_RESET'; LibVersion := '9.0' } : MC_RESET;
      instReset_Kin { InstructionName := 'MC_RESET'; LibVersion := '9.0' } : MC_RESET;
   END_VAR


BEGIN

	// =====================================================================
	// REGION Power — per-axis MC_Power calls
	// All 4 joints share the same enableAxes bit + StartMode[i]/StopMode[i].
	// =====================================================================
	#instPower_J1(Axis      := "J1_SCARA_Arm3D",
	              Enable    := "GDB_Control".enableAxes,
	              StartMode := "GDB_Control".StartMode[1],
	              StopMode  := "GDB_Control".StopMode[1]);

	#instPower_J2(Axis      := "J2_SCARA_Arm3D",
	              Enable    := "GDB_Control".enableAxes,
	              StartMode := "GDB_Control".StartMode[2],
	              StopMode  := "GDB_Control".StopMode[2]);

	#instPower_J3(Axis      := "J3_SCARA_Arm3D",
	              Enable    := "GDB_Control".enableAxes,
	              StartMode := "GDB_Control".StartMode[3],
	              StopMode  := "GDB_Control".StopMode[3]);

	#instPower_J4(Axis      := "J4_SCARA_Arm3D",
	              Enable    := "GDB_Control".enableAxes,
	              StartMode := "GDB_Control".StartMode[4],
	              StopMode  := "GDB_Control".StopMode[4]);

	// Mirror axesEnabled = AND of all 4 Status outputs
	"GDB_Control".axesEnabled := #instPower_J1.Status
	                              AND #instPower_J2.Status
	                              AND #instPower_J3.Status
	                              AND #instPower_J4.Status;

	// =====================================================================
	// REGION Reset — 4 per-axis MC_RESET + 1 on kinematic TO
	// MC_RESET accepts TO_PositioningAxis (joints) AND TO_Kinematics (group).
	// Single rising-edge from HMI resetAxes button.
	// =====================================================================
	#instReset_J1(Axis := "J1_SCARA_Arm3D", Execute := "GDB_Control".resetAxes);
	#instReset_J2(Axis := "J2_SCARA_Arm3D", Execute := "GDB_Control".resetAxes);
	#instReset_J3(Axis := "J3_SCARA_Arm3D", Execute := "GDB_Control".resetAxes);
	#instReset_J4(Axis := "J4_SCARA_Arm3D", Execute := "GDB_Control".resetAxes);
	#instReset_Kin(Axis := "ScaraArm3D",    Execute := "GDB_Control".resetAxes);

	"GDB_Control".axesError := #instPower_J1.Error
	                            OR #instPower_J2.Error
	                            OR #instPower_J3.Error
	                            OR #instPower_J4.Error
	                            OR #instHome_J1.Error
	                            OR #instHome_J2.Error
	                            OR #instHome_J3.Error
	                            OR #instHome_J4.Error
	                            OR #instReset_J1.Error
	                            OR #instReset_J2.Error
	                            OR #instReset_J3.Error
	                            OR #instReset_J4.Error
	                            OR #instReset_Kin.Error;

	// =====================================================================
	// REGION Home — per-axis MC_Home calls
	// HomeMode[i]=7 ("set actual position") — no physical homing motion.
	// HomePos[i] from Startup OB (all zeros for SCARA zero pose).
	// =====================================================================
	#instHome_J1(Axis     := "J1_SCARA_Arm3D",
	             Execute  := "GDB_Control".homeAxes,
	             Position := "GDB_Control".HomePos[1],
	             Mode     := "GDB_Control".HomeMode[1]);

	#instHome_J2(Axis     := "J2_SCARA_Arm3D",
	             Execute  := "GDB_Control".homeAxes,
	             Position := "GDB_Control".HomePos[2],
	             Mode     := "GDB_Control".HomeMode[2]);

	#instHome_J3(Axis     := "J3_SCARA_Arm3D",
	             Execute  := "GDB_Control".homeAxes,
	             Position := "GDB_Control".HomePos[3],
	             Mode     := "GDB_Control".HomeMode[3]);

	#instHome_J4(Axis     := "J4_SCARA_Arm3D",
	             Execute  := "GDB_Control".homeAxes,
	             Position := "GDB_Control".HomePos[4],
	             Mode     := "GDB_Control".HomeMode[4]);

	// Mirror axesHomed = AND of all 4 Done outputs
	IF #instHome_J1.Done
	   AND #instHome_J2.Done
	   AND #instHome_J3.Done
	   AND #instHome_J4.Done
	THEN
	    "GDB_Control".axesHomed := TRUE;
	END_IF;

END_FUNCTION_BLOCK

FUNCTION_BLOCK "FB_ConveyorCtrl"
{ S7_Optimized_Access := 'TRUE' }
VERSION : 1.3
// =====================================================================
// FB_ConveyorCtrl  V1.3  (2026-05-20)
// V1.3: belt-stop is LEVEL-triggered on PalletizingSensor, not its edge.
//       An edge-RESET missed a box already at the pick end when the
//       cycle started -> belt ran forever (Belt=200, sensor TRUE, 90 s).
// V1.2: belt now starts at SPAWN, not at PackingSensor (the box spawns
//       upstream of PackingSensor; waiting for it deadlocked).
// V1.1: spawn pulse widened 100 ms -> 2 s for reliable co-sim edge catch.
// ---------------------------------------------------------------------
// Owns the palletizing INFEED: the box-spawn request (SpawnContainerCmd)
// and the conveyor belt (BeltVelocity). Splitting this out of
// FB_AutoCtrl_Palletizing leaves the palletizer as pure pick-and-place.
//
// Runs in REAL mode only (GDB_PalletizingCmd.bo_RequireSensorGate=TRUE).
// In phantom mode it never starts and simply holds SpawnContainerCmd =
// FALSE and BeltVelocity = 0 every scan -- it is the SOLE writer of both,
// so it must drive them to a defined value at all times.
//
// Box flow it paces, x16:
//   spawn pulse          -> belt starts + NX spawns 1 box at the origin
//   ~belt transit        -> box rides the belt past PackingSensor
//   PalletizingSensor ^  -> belt stops (SCARA picks the box)
//   PalletizingSensor v  -> box picked away -> request the next box
//
// No MC instructions -> zero OB91 (MC-Servo) impact. Raw R_TRIG /
// F_TRIG / TON_TIME + DB writes only -- no libraries (gate V1).
//
// Coordination with FB_AutoCtrl_Palletizing: no direct FB-to-FB signal.
// Both FBs start/stop on the same GDB_PalletizingCmd command bits; the
// two belt sensors are the runtime handshake. The conveyor presents a
// box at PalletizingSensor, the palletizer's WAIT_ARRIVAL picks it, the
// pick clears PalletizingSensor, the conveyor spawns the next. The two
// independent counts (conveyor spawns 16, palletizer places 16) stay in
// lockstep through the physical one-box-at-a-time flow.
// =====================================================================
// Edge-detect instances
   VAR 
      sRTRIGStart {InstructionName := 'R_TRIG'; LibVersion := '1.0'} : R_TRIG;
      sRTRIGStop {InstructionName := 'R_TRIG'; LibVersion := '1.0'} : R_TRIG;
      sRTRIGPacking {InstructionName := 'R_TRIG'; LibVersion := '1.0'} : R_TRIG;
      sRTRIGPalletizing {InstructionName := 'R_TRIG'; LibVersion := '1.0'} : R_TRIG;
      sFTRIGPalletizing {InstructionName := 'F_TRIG'; LibVersion := '1.0'} : F_TRIG;
      sRTRIGSpawnFire {InstructionName := 'R_TRIG'; LibVersion := '1.0'} : R_TRIG;   // Spawn-pulse timer
      instSpawnTimer {InstructionName := 'TON_TIME'; LibVersion := '1.0'} : TON_TIME;   // State
      statRunning : Bool;   // TRUE between Start and Stop (real mode only)
      statSpawnFire : Bool;   // one-shot spawn request (rising edge -> one pulse)
      statSpawnActive : Bool;   // TRUE while the spawn pulse is in flight
      statBeltRun : Bool;   // belt latch: SET by PackingSensor, RESET by PalletizingSensor
      statSpawnCount : Int;   // boxes requested so far this run (capped at i16_TotalBoxes)
   END_VAR


BEGIN
	
	
	 // =====================================================================
	 // REGION 1 -- EDGE DETECTORS
	 // =====================================================================
	 #sRTRIGStart(CLK := "GDB_PalletizingCmd".bo_Start);
	 #sRTRIGStop(CLK := "GDB_PalletizingCmd".bo_Stop);
	 #sRTRIGPacking(CLK := "GDB_MCDData".PackingSensor);
	 #sRTRIGPalletizing(CLK := "GDB_MCDData".PalletizingSensor);
	 #sFTRIGPalletizing(CLK := "GDB_MCDData".PalletizingSensor);
	
	 // =====================================================================
	 // REGION 2 -- START
	 // Lockstep with FB_AutoCtrl_Palletizing REGION 2: the conveyor starts
	 // under exactly the conditions the palletizer starts, plus
	 // bo_RequireSensorGate (conveyor is real-mode only) and NOT statRunning
	 // (idle guard -- the conveyor analog of the palletizer i16_PalletStep=0).
	 // =====================================================================
	 IF #sRTRIGStart.Q
	     AND "GDB_PalletizingCmd".bo_Mode
	     AND "GDB_PalletizingCmd".bo_RequireSensorGate
	     AND "GDB_PalletizingCmd".bo_ESTOP_LOCK
	     AND "GDB_PalletizingCmd".bo_PalletInitialed
	     AND NOT "GDB_PalletizingCmd".bo_Alarm
	     AND NOT "GDB_MachineCmd".bo_Mode
	     AND NOT "GDB_ManualCmd".bo_Mode
	     AND NOT #statRunning
	 THEN
	     #statRunning    := TRUE;
	     #statSpawnCount := 0;
	     #statBeltRun    := FALSE;
	     #statSpawnFire  := TRUE;     // request box 1
	 END_IF;
	
	 // =====================================================================
	 // REGION 3 -- STOP  (bo_Stop edge, alarm latched, or left real mode)
	 // =====================================================================
	 IF #sRTRIGStop.Q
	     OR "GDB_PalletizingCmd".bo_Alarm
	     OR NOT "GDB_PalletizingCmd".bo_RequireSensorGate
	 THEN
	     #statRunning     := FALSE;
	     #statBeltRun     := FALSE;
	     #statSpawnFire   := FALSE;
	     #statSpawnActive := FALSE;
	 END_IF;
	
	 // =====================================================================
	 // REGION 4 -- SPAWN PACING
	 // One box at a time: request the next only once the previous has been
	 // picked away (PalletizingSensor falling edge). statSpawnCount caps the
	 // run at i16_TotalBoxes total spawns -- a stray sensor drop can mistime
	 // a spawn but can never spawn more than i16_TotalBoxes boxes.
	 // =====================================================================
	 IF #sFTRIGPalletizing.Q
	     AND #statRunning
	     AND (#statSpawnCount < "GDB_PalletizingCmd".i16_TotalBoxes)
	 THEN
	     #statSpawnFire := TRUE;
	 END_IF;
	
	 // =====================================================================
	 // REGION 5 -- SPAWN-PULSE GENERATOR  (SOLE writer of SpawnContainerCmd)
	 // sRTRIGSpawnFire arms a pulse on the RISING EDGE of statSpawnFire, so a
	 // stuck-TRUE request still yields at most one pulse, never a train.
	 // Pulse width 2 s -- long enough for the NX MCD co-sim to reliably
	 // catch the rising edge. objsrcContainer "Once per Activation" spawns
	 // exactly one box per rising edge regardless of how long active is
	 // held (trace-confirmed). statSpawnCount += 1 per armed pulse.
	 // The belt is ALSO started here -- the box spawns upstream of
	 // PackingSensor, so the belt must run from the spawn to carry the box
	 // onto the sensor; waiting for PackingSensor to start it deadlocks.
	 // =====================================================================
	 #sRTRIGSpawnFire(CLK := #statSpawnFire);
	 IF #sRTRIGSpawnFire.Q THEN
	     #statSpawnActive := TRUE;
	     #statSpawnCount  := #statSpawnCount + 1;
	     #statBeltRun     := TRUE;
	 END_IF;
	
	 IF #statSpawnActive THEN
	     "GDB_MCDData".SpawnContainerCmd := TRUE;
	     #instSpawnTimer(IN := TRUE, PT := T#2S);
	     IF #instSpawnTimer.Q THEN
	         "GDB_MCDData".SpawnContainerCmd := FALSE;
	         #instSpawnTimer(IN := FALSE, PT := T#0MS);
	         #statSpawnActive := FALSE;
	         #statSpawnFire   := FALSE;
	     END_IF;
	 ELSE
	     "GDB_MCDData".SpawnContainerCmd := FALSE;
	     #instSpawnTimer(IN := FALSE, PT := T#0MS);
	 END_IF;
	
	 // =====================================================================
	 // REGION 6 -- BELT LATCH + OUTPUT  (SOLE writer of BeltVelocity)
	 // statBeltRun is SET at spawn (REGION 5); PackingSensor rising re-SETs
	 // it as redundant confirmation. It is RESET on the LEVEL of
	 // PalletizingSensor -- the belt stops whenever a box is at the pick
	 // end, even if that box was already there before the cycle began. An
	 // edge-RESET missed an already-TRUE sensor and the belt never stopped.
	 // =====================================================================
	 IF #sRTRIGPacking.Q THEN
	     #statBeltRun := TRUE;
	 END_IF;
	 IF "GDB_MCDData".PalletizingSensor THEN
	     #statBeltRun := FALSE;
	 END_IF;
	
	 IF #statRunning AND #statBeltRun THEN
	     "GDB_MCDData".BeltVelocity := "GDB_PalletizingCmd".lr_BeltVelocityNormal;
	 ELSE
	     "GDB_MCDData".BeltVelocity := 0.0;
	 END_IF;
	
	
END_FUNCTION_BLOCK

FUNCTION_BLOCK "FB_ManualCtrl"
{ S7_Optimized_Access := 'TRUE' }
VERSION : 1.2
// =====================================================================
// SCARA ABCDE - Manual Control Surface  (Phase 5, 2026-05-21)
//
// Runs in OB1 (process logic). Routes HMI manual-mode commands
// (GDB_ManualCmd) to the 600 axis layer by WRITING GDB_AxisCtrl - it
// never calls an MC instruction.
//   REGION Mode_Gate              - compute statManualOK (mutex + safety)
//   REGION Group_Enable_Home_Reset- Enable/Home/Reset -> GDB_AxisCtrl input
//   REGION Cartesian_Jog          - HMI jog buttons -> ...input.jogframe;
//                                   FB_AxisCtrl (OB30) runs LKinCtrl_MC_JogFrame.
//   REGION Kin_Manual_Move        - bo_KinGo -> ...input.movelinear (the same
//                                   interface the auto FBs use).
//   REGION Status_Mirror          - TO StatusWord + GDB_AxisCtrl -> GDB_ManualStatus
//
// V1.2 (2026-05-22) - Task #5: REGION Group_Enable_Home_Reset stands down while
// FB_AxisCtrl's guided recovery runs (GDB_AxisCtrl.LKinCtrl.output.bo_recovering),
// so the recovery sequencer is the single writer of input.bo_enable/home/reset.
// V1.1 (2026-05-22) - REGION Kin_Manual_Move sets input.movelinear.bo_isPTP
// := FALSE so manual moves stay Cartesian linear (FB_AxisCtrl V2.3 added a
// PTP route on that shared bit for the palletizing transits).
// V1.0 (Phase 5) - rebuilt: the 4x MC_MoveJog and the 1x MC_MoveLinear-
// Absolute are removed. MC_MoveJog conflicts with axes inside a kinematics
// group, so jog now goes through LKinCtrl_MC_JogFrame in the OB30 layer.
//
// Jog is CARTESIAN (WCS): the HMI's 4 jog axis-pairs drive the TCP in
// X / Y / Z / A. The bo_J{n}_Jog* button names are legacy - the Phase 6
// HMI update relabels them X/Y/Z/A.
//
// Mutex: statManualOK := bo_Mode AND bo_ESTOP_LOCK AND NOT
// GDB_MachineCmd.bo_Mode. When FALSE, REGIONs 2-4 make no motion writes
// (jog bits forced FALSE); REGION Status_Mirror always runs.
// =====================================================================
   VAR
      sRTRIGKinGo {InstructionName := 'R_TRIG'; LibVersion := '1.0'} : R_TRIG;
      statManualOK : Bool;
   END_VAR

   VAR_TEMP
      tempEnableAxes : Bool;
      tempHomeAxes : Bool;
      tempResetAxes : Bool;
   END_VAR


BEGIN

    REGION Mode_Gate
        // statManualOK gates the routing regions. Mutex with the auto FBs:
        // manual requires ABCDE auto mode (GDB_MachineCmd.bo_Mode) is FALSE.
        #statManualOK := "GDB_ManualCmd".bo_Mode
                         AND "GDB_ManualCmd".bo_ESTOP_LOCK
                         AND NOT "GDB_MachineCmd".bo_Mode;
    END_REGION

    REGION Group_Enable_Home_Reset
        // Per-axis + Kin-group Enable/Home/Reset buttons OR into the shared
        // GDB_AxisCtrl group request bits. FB_AxisCtrl (OB30) drives the
        // LKinCtrl group power / reset; FB_Init drives the homing. Per-axis
        // is a UX nicety - enable/home/reset are group-level. Task #5: while
        // FB_AxisCtrl's guided recovery runs (output.bo_recovering), it owns
        // these bits - this region stands down so there is a single writer.
        IF #statManualOK AND NOT "GDB_AxisCtrl".LKinCtrl.output.bo_recovering THEN
            #tempEnableAxes := "GDB_ManualCmd".bo_J1_Enable
                               OR "GDB_ManualCmd".bo_J2_Enable
                               OR "GDB_ManualCmd".bo_J3_Enable
                               OR "GDB_ManualCmd".bo_J4_Enable
                               OR "GDB_ManualCmd".bo_KinEnable;
            #tempHomeAxes := "GDB_ManualCmd".bo_J1_Home
                             OR "GDB_ManualCmd".bo_J2_Home
                             OR "GDB_ManualCmd".bo_J3_Home
                             OR "GDB_ManualCmd".bo_J4_Home
                             OR "GDB_ManualCmd".bo_KinHome;
            #tempResetAxes := "GDB_ManualCmd".bo_J1_Reset
                              OR "GDB_ManualCmd".bo_J2_Reset
                              OR "GDB_ManualCmd".bo_J3_Reset
                              OR "GDB_ManualCmd".bo_J4_Reset
                              OR "GDB_ManualCmd".bo_KinReset;

            "GDB_AxisCtrl".LKinCtrl.input.bo_enable := #tempEnableAxes;
            "GDB_AxisCtrl".LKinCtrl.input.bo_home   := #tempHomeAxes;
            "GDB_AxisCtrl".LKinCtrl.input.bo_reset  := #tempResetAxes;
        END_IF;
    END_REGION

